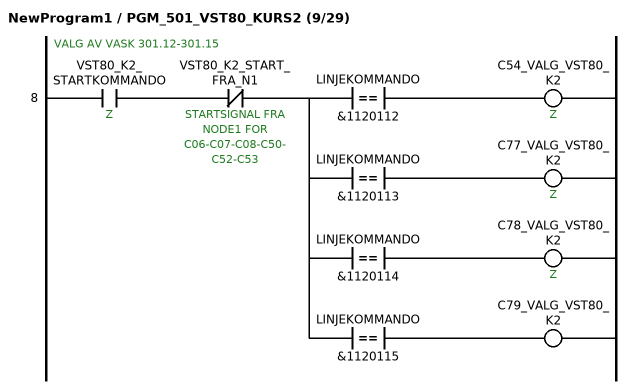
; [picture p504: NewProgram1 / PGM_501_VST80_KURS2, rungs 8-8]
; rung 8: VALG AV VASK 301.12-301.15
LD VST80_K2_STARTKOMMANDO  ; Z
ANDNOT VST80_K2_START_FRA_N1  ; STARTSIGNAL FRA NODE1 FOR C06-C07-C08-C50-C52-C53
OUT TR0
AND=L(301) LINJEKOMMANDO &1120112
OUT C54_VALG_VST80_K2  ; Z
LD TR0
AND=L(301) LINJEKOMMANDO &1120113
OUT C77_VALG_VST80_K2  ; Z
LD TR0
AND=L(301) LINJEKOMMANDO &1120114
OUT C78_VALG_VST80_K2  ; Z
LD TR0
AND=L(301) LINJEKOMMANDO &1120115
OUT C79_VALG_VST80_K2

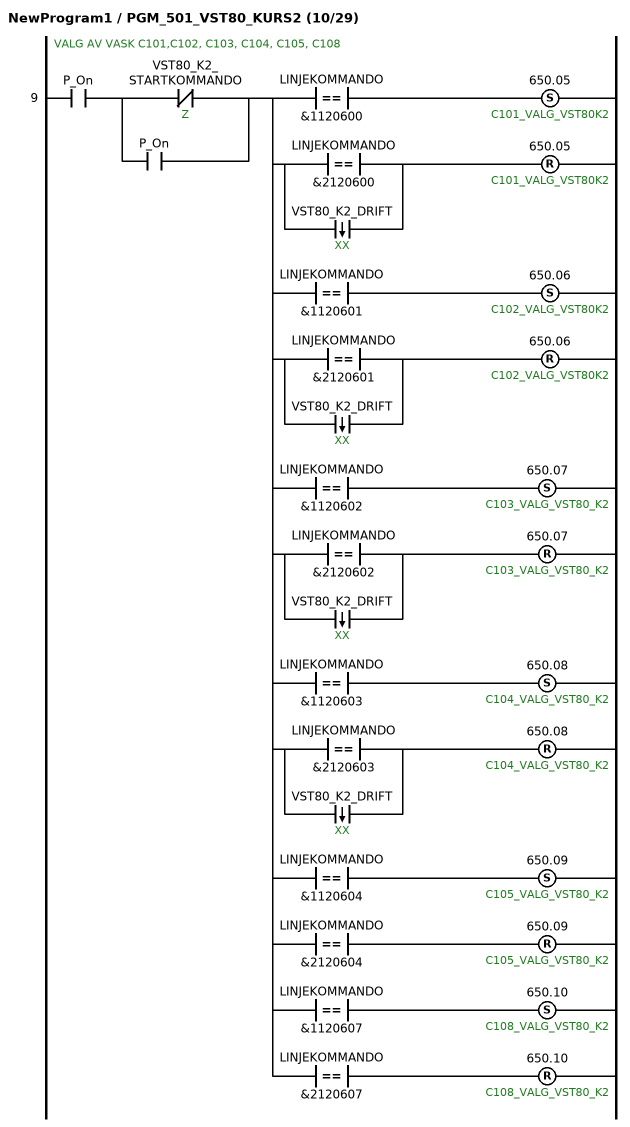
; rung 9: VALG AV VASK C101,C102, C103, C104, C105, C108
LD P_On
LDNOT VST80_K2_STARTKOMMANDO  ; Z
OR P_On
ANDLD
OUT TR0
AND=L(301) LINJEKOMMANDO &1120600
SET 650.05  ; C101_VALG_VST80K2
LD TR0
LD=L(301) LINJEKOMMANDO &2120600
%OR VST80_K2_DRIFT  ; XX
ANDLD
RSET 650.05  ; C101_VALG_VST80K2
LD TR0
AND=L(301) LINJEKOMMANDO &1120601
SET 650.06  ; C102_VALG_VST80K2
LD TR0
LD=L(301) LINJEKOMMANDO &2120601
%OR VST80_K2_DRIFT  ; XX
ANDLD
RSET 650.06  ; C102_VALG_VST80K2
LD TR0
AND=L(301) LINJEKOMMANDO &1120602
SET 650.07  ; C103_VALG_VST80_K2
LD TR0
LD=L(301) LINJEKOMMANDO &2120602
%OR VST80_K2_DRIFT  ; XX
ANDLD
RSET 650.07  ; C103_VALG_VST80_K2
LD TR0
AND=L(301) LINJEKOMMANDO &1120603
SET 650.08  ; C104_VALG_VST80_K2
LD TR0
LD=L(301) LINJEKOMMANDO &2120603
%OR VST80_K2_DRIFT  ; XX
ANDLD
RSET 650.08  ; C104_VALG_VST80_K2
LD TR0
AND=L(301) LINJEKOMMANDO &1120604
SET 650.09  ; C105_VALG_VST80_K2
LD TR0
AND=L(301) LINJEKOMMANDO &2120604
RSET 650.09  ; C105_VALG_VST80_K2
LD TR0
AND=L(301) LINJEKOMMANDO &1120607
SET 650.10  ; C108_VALG_VST80_K2
LD TR0
AND=L(301) LINJEKOMMANDO &2120607
RSET 650.10  ; C108_VALG_VST80_K2

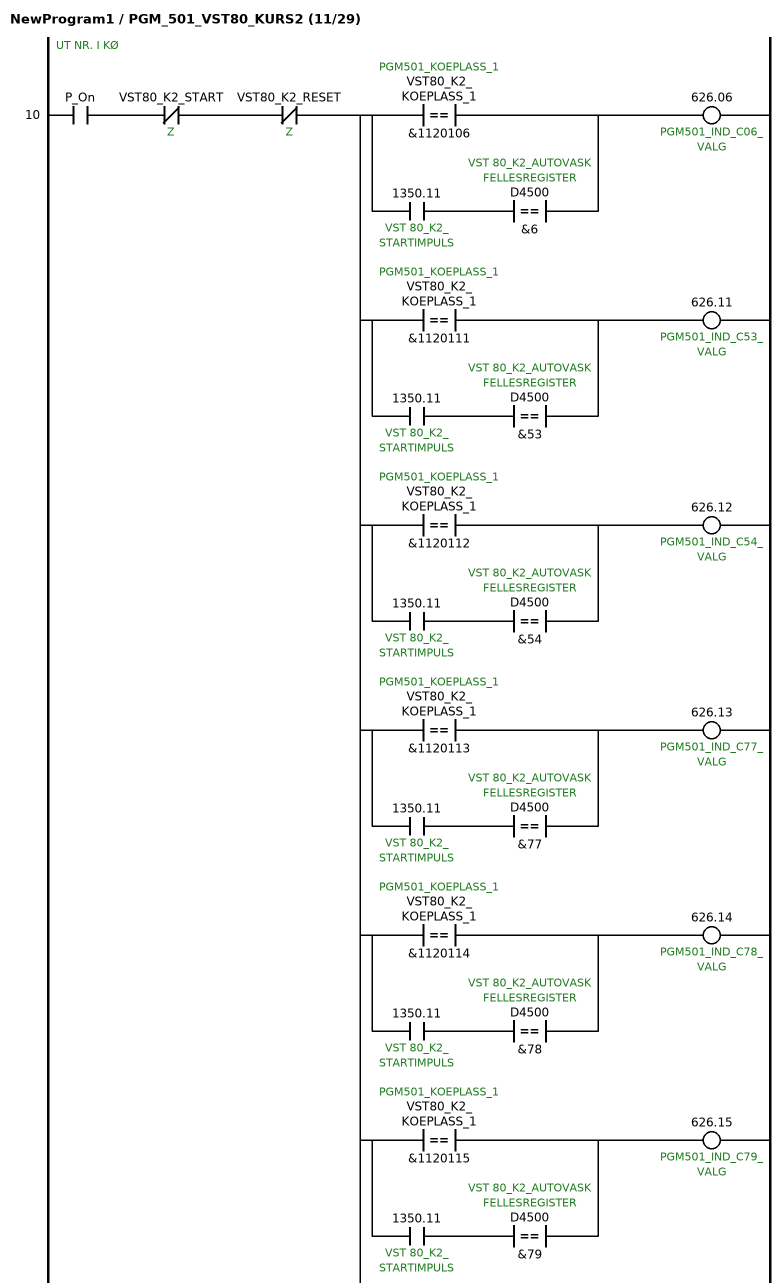

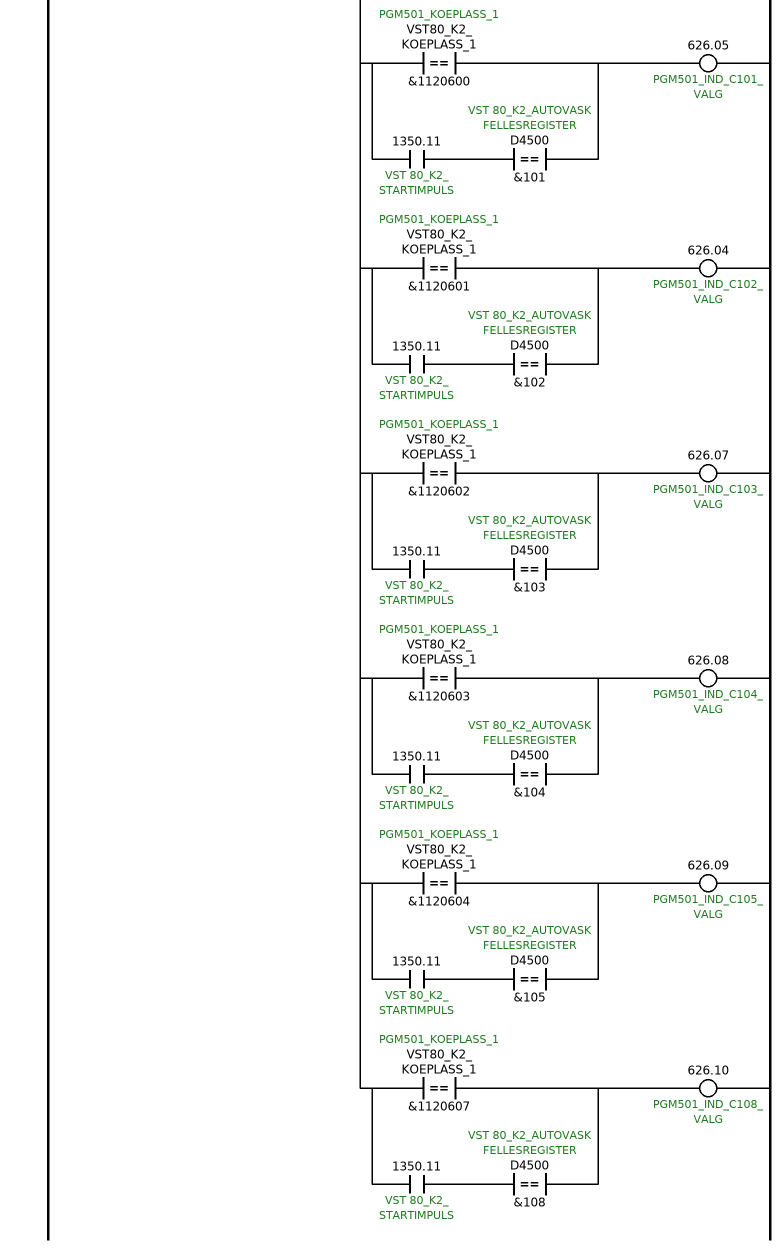
; rung 10: UT NR. I KØ
LD P_On
ANDNOT VST80_K2_START  ; Z
ANDNOT VST80_K2_RESET  ; Z
OUT TR0
LD=L(301) VST80_K2_KOEPLASS_1 &1120106  ; PGM501_KOEPLASS_1
LD 1350.11  ; VST 80_K2_STARTIMPULS
AND=(300) D4500 &6  ; VST 80_K2_AUTOVASK FELLESREGISTER
ORLD
ANDLD
OUT 626.06  ; PGM501_IND_C06_VALG
LD TR0
LD=L(301) VST80_K2_KOEPLASS_1 &1120111  ; PGM501_KOEPLASS_1
LD 1350.11  ; VST 80_K2_STARTIMPULS
AND=(300) D4500 &53  ; VST 80_K2_AUTOVASK FELLESREGISTER
ORLD
ANDLD
OUT 626.11  ; PGM501_IND_C53_VALG
LD TR0
LD=L(301) VST80_K2_KOEPLASS_1 &1120112  ; PGM501_KOEPLASS_1
LD 1350.11  ; VST 80_K2_STARTIMPULS
AND=(300) D4500 &54  ; VST 80_K2_AUTOVASK FELLESREGISTER
ORLD
ANDLD
OUT 626.12  ; PGM501_IND_C54_VALG
LD TR0
LD=L(301) VST80_K2_KOEPLASS_1 &1120113  ; PGM501_KOEPLASS_1
LD 1350.11  ; VST 80_K2_STARTIMPULS
AND=(300) D4500 &77  ; VST 80_K2_AUTOVASK FELLESREGISTER
ORLD
ANDLD
OUT 626.13  ; PGM501_IND_C77_VALG
LD TR0
LD=L(301) VST80_K2_KOEPLASS_1 &1120114  ; PGM501_KOEPLASS_1
LD 1350.11  ; VST 80_K2_STARTIMPULS
AND=(300) D4500 &78  ; VST 80_K2_AUTOVASK FELLESREGISTER
ORLD
ANDLD
OUT 626.14  ; PGM501_IND_C78_VALG
LD TR0
LD=L(301) VST80_K2_KOEPLASS_1 &1120115  ; PGM501_KOEPLASS_1
LD 1350.11  ; VST 80_K2_STARTIMPULS
AND=(300) D4500 &79  ; VST 80_K2_AUTOVASK FELLESREGISTER
ORLD
ANDLD
OUT 626.15  ; PGM501_IND_C79_VALG
LD TR0
LD=L(301) VST80_K2_KOEPLASS_1 &1120600  ; PGM501_KOEPLASS_1
LD 1350.11  ; VST 80_K2_STARTIMPULS
AND=(300) D4500 &101  ; VST 80_K2_AUTOVASK FELLESREGISTER
ORLD
ANDLD
OUT 626.05  ; PGM501_IND_C101_VALG
LD TR0
LD=L(301) VST80_K2_KOEPLASS_1 &1120601  ; PGM501_KOEPLASS_1
LD 1350.11  ; VST 80_K2_STARTIMPULS
AND=(300) D4500 &102  ; VST 80_K2_AUTOVASK FELLESREGISTER
ORLD
ANDLD
OUT 626.04  ; PGM501_IND_C102_VALG
LD TR0
LD=L(301) VST80_K2_KOEPLASS_1 &1120602  ; PGM501_KOEPLASS_1
LD 1350.11  ; VST 80_K2_STARTIMPULS
AND=(300) D4500 &103  ; VST 80_K2_AUTOVASK FELLESREGISTER
ORLD
ANDLD
OUT 626.07  ; PGM501_IND_C103_VALG
LD TR0
LD=L(301) VST80_K2_KOEPLASS_1 &1120603  ; PGM501_KOEPLASS_1
LD 1350.11  ; VST 80_K2_STARTIMPULS
AND=(300) D4500 &104  ; VST 80_K2_AUTOVASK FELLESREGISTER
ORLD
ANDLD
OUT 626.08  ; PGM501_IND_C104_VALG
LD TR0
LD=L(301) VST80_K2_KOEPLASS_1 &1120604  ; PGM501_KOEPLASS_1
LD 1350.11  ; VST 80_K2_STARTIMPULS
AND=(300) D4500 &105  ; VST 80_K2_AUTOVASK FELLESREGISTER
ORLD
ANDLD
OUT 626.09  ; PGM501_IND_C105_VALG
LD TR0
LD=L(301) VST80_K2_KOEPLASS_1 &1120607  ; PGM501_KOEPLASS_1
LD 1350.11  ; VST 80_K2_STARTIMPULS
AND=(300) D4500 &108  ; VST 80_K2_AUTOVASK FELLESREGISTER
ORLD
ANDLD
OUT 626.10  ; PGM501_IND_C108_VALG

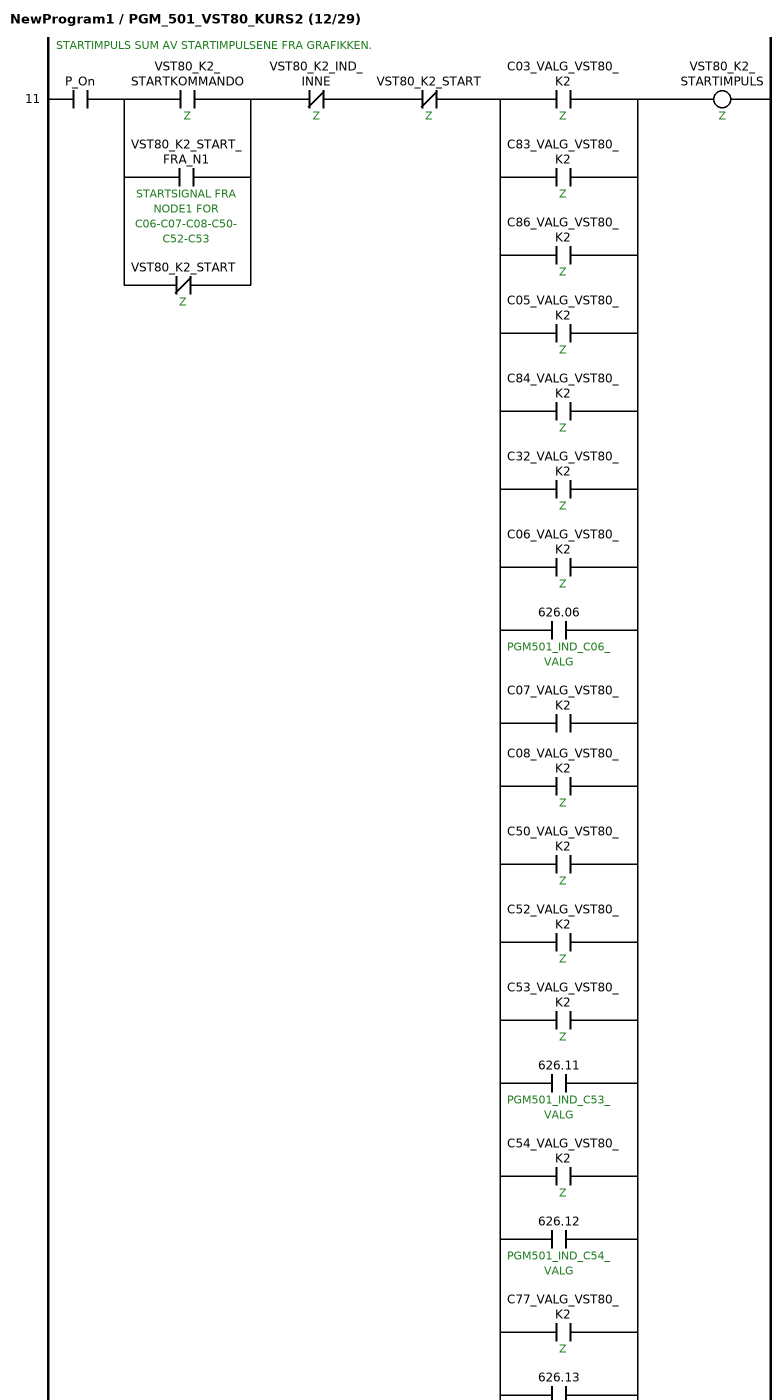

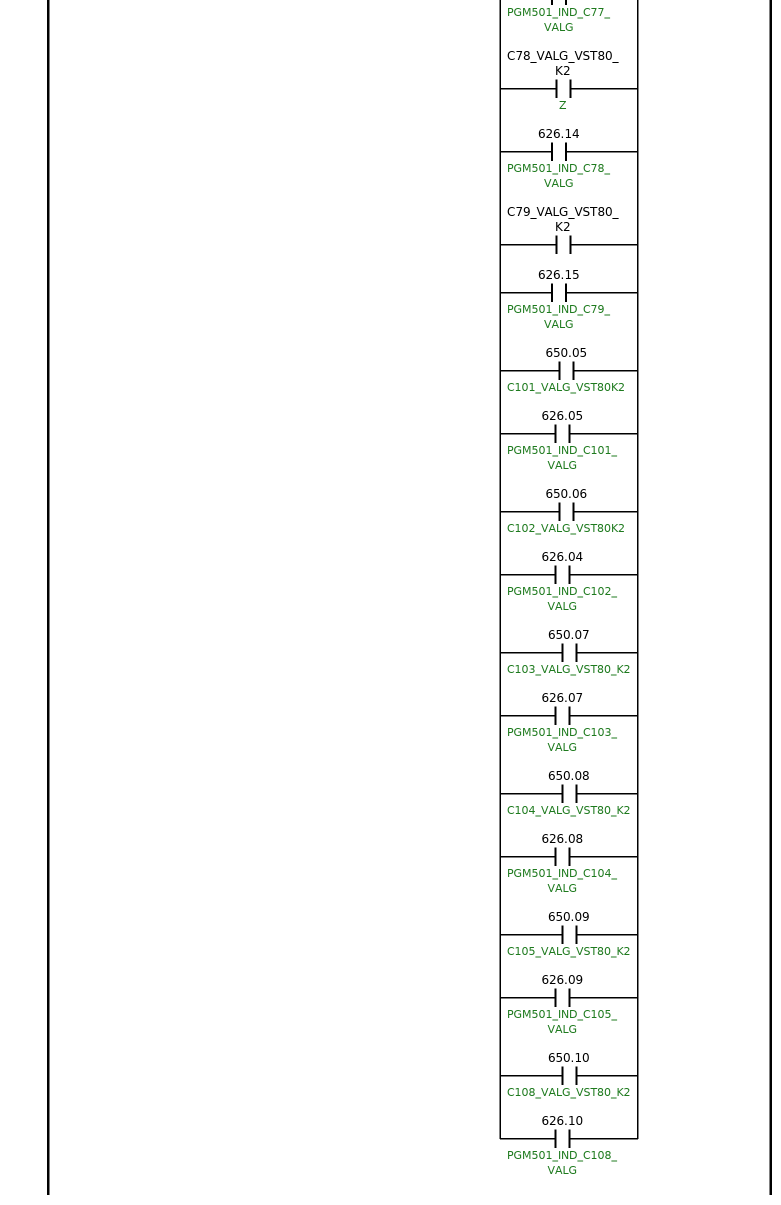
; rung 11: STARTIMPULS SUM AV STARTIMPULSENE FRA GRAFIKKEN.
LD P_On
LD VST80_K2_STARTKOMMANDO  ; Z
OR VST80_K2_START_FRA_N1  ; STARTSIGNAL FRA NODE1 FOR C06-C07-C08-C50-C52-C53
ORNOT VST80_K2_START  ; Z
ANDLD
ANDNOT VST80_K2_IND_INNE  ; Z
ANDNOT VST80_K2_START  ; Z
LD C03_VALG_VST80_K2  ; Z
OR C83_VALG_VST80_K2  ; Z
OR C86_VALG_VST80_K2  ; Z
OR C05_VALG_VST80_K2  ; Z
OR C84_VALG_VST80_K2  ; Z
OR C32_VALG_VST80_K2  ; Z
OR C06_VALG_VST80_K2  ; Z
OR 626.06  ; PGM501_IND_C06_VALG
OR C07_VALG_VST80_K2
OR C08_VALG_VST80_K2  ; Z
OR C50_VALG_VST80_K2  ; Z
OR C52_VALG_VST80_K2  ; Z
OR C53_VALG_VST80_K2  ; Z
OR 626.11  ; PGM501_IND_C53_VALG
OR C54_VALG_VST80_K2  ; Z
OR 626.12  ; PGM501_IND_C54_VALG
OR C77_VALG_VST80_K2  ; Z
OR 626.13  ; PGM501_IND_C77_VALG
OR C78_VALG_VST80_K2  ; Z
OR 626.14  ; PGM501_IND_C78_VALG
OR C79_VALG_VST80_K2
OR 626.15  ; PGM501_IND_C79_VALG
OR 650.05  ; C101_VALG_VST80K2
OR 626.05  ; PGM501_IND_C101_VALG
OR 650.06  ; C102_VALG_VST80K2
OR 626.04  ; PGM501_IND_C102_VALG
OR 650.07  ; C103_VALG_VST80_K2
OR 626.07  ; PGM501_IND_C103_VALG
OR 650.08  ; C104_VALG_VST80_K2
OR 626.08  ; PGM501_IND_C104_VALG
OR 650.09  ; C105_VALG_VST80_K2
OR 626.09  ; PGM501_IND_C105_VALG
OR 650.10  ; C108_VALG_VST80_K2
OR 626.10  ; PGM501_IND_C108_VALG
ANDLD
OUT VST80_K2_STARTIMPULS  ; Z

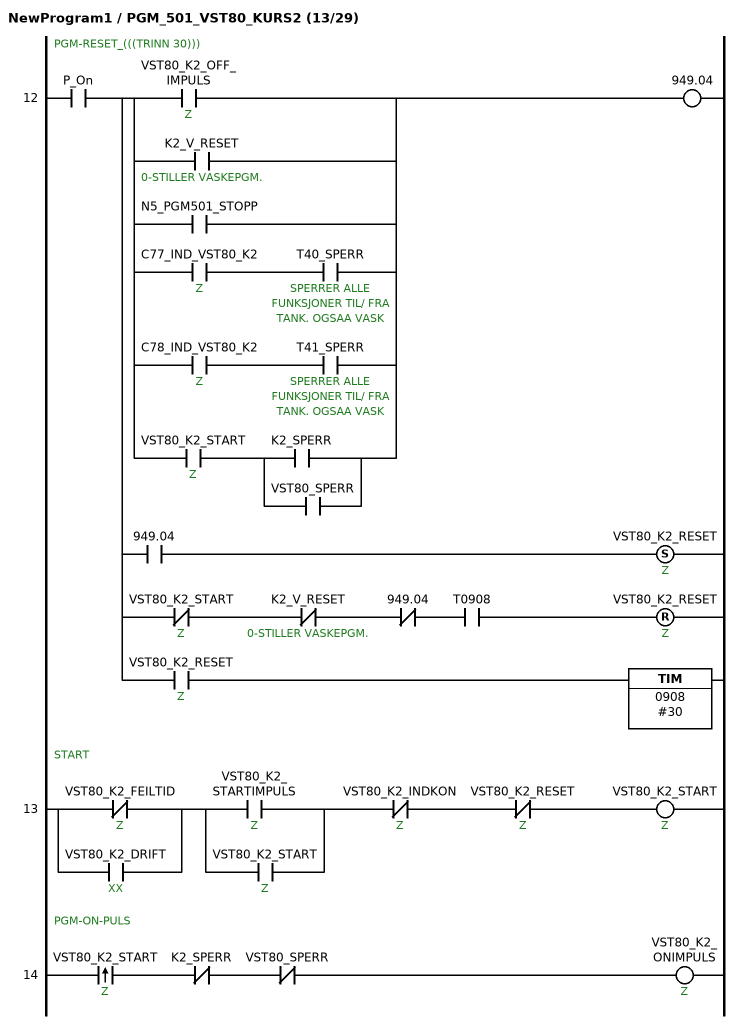
; rung 12: PGM-RESET_(((TRINN 30)))
LD P_On
OUT TR0
LD VST80_K2_OFF_IMPULS  ; Z
OR K2_V_RESET  ; 0-STILLER VASKEPGM.
OR N5_PGM501_STOPP
LD C77_IND_VST80_K2  ; Z
AND T40_SPERR  ; SPERRER ALLE FUNKSJONER TIL/ FRA TANK. OGSAA VASK
ORLD
LD C78_IND_VST80_K2  ; Z
AND T41_SPERR  ; SPERRER ALLE FUNKSJONER TIL/ FRA TANK. OGSAA VASK
ORLD
LD VST80_K2_START  ; Z
LD K2_SPERR
OR VST80_SPERR
ANDLD
ORLD
ANDLD
OUT 949.04
LD TR0
AND 949.04
SET VST80_K2_RESET  ; Z
LD TR0
ANDNOT VST80_K2_START  ; Z
ANDNOT K2_V_RESET  ; 0-STILLER VASKEPGM.
ANDNOT 949.04
AND T0908
RSET VST80_K2_RESET  ; Z
LD TR0
AND VST80_K2_RESET  ; Z
TIM 0908 #30
; rung 13: START
LDNOT VST80_K2_FEILTID  ; Z
OR VST80_K2_DRIFT  ; XX
LD VST80_K2_STARTIMPULS  ; Z
OR VST80_K2_START  ; Z
ANDLD
ANDNOT VST80_K2_INDKON  ; Z
ANDNOT VST80_K2_RESET  ; Z
OUT VST80_K2_START  ; Z
; rung 14: PGM-ON-PULS
@LD VST80_K2_START  ; Z
ANDNOT K2_SPERR
ANDNOT VST80_SPERR
OUT VST80_K2_ONIMPULS  ; Z

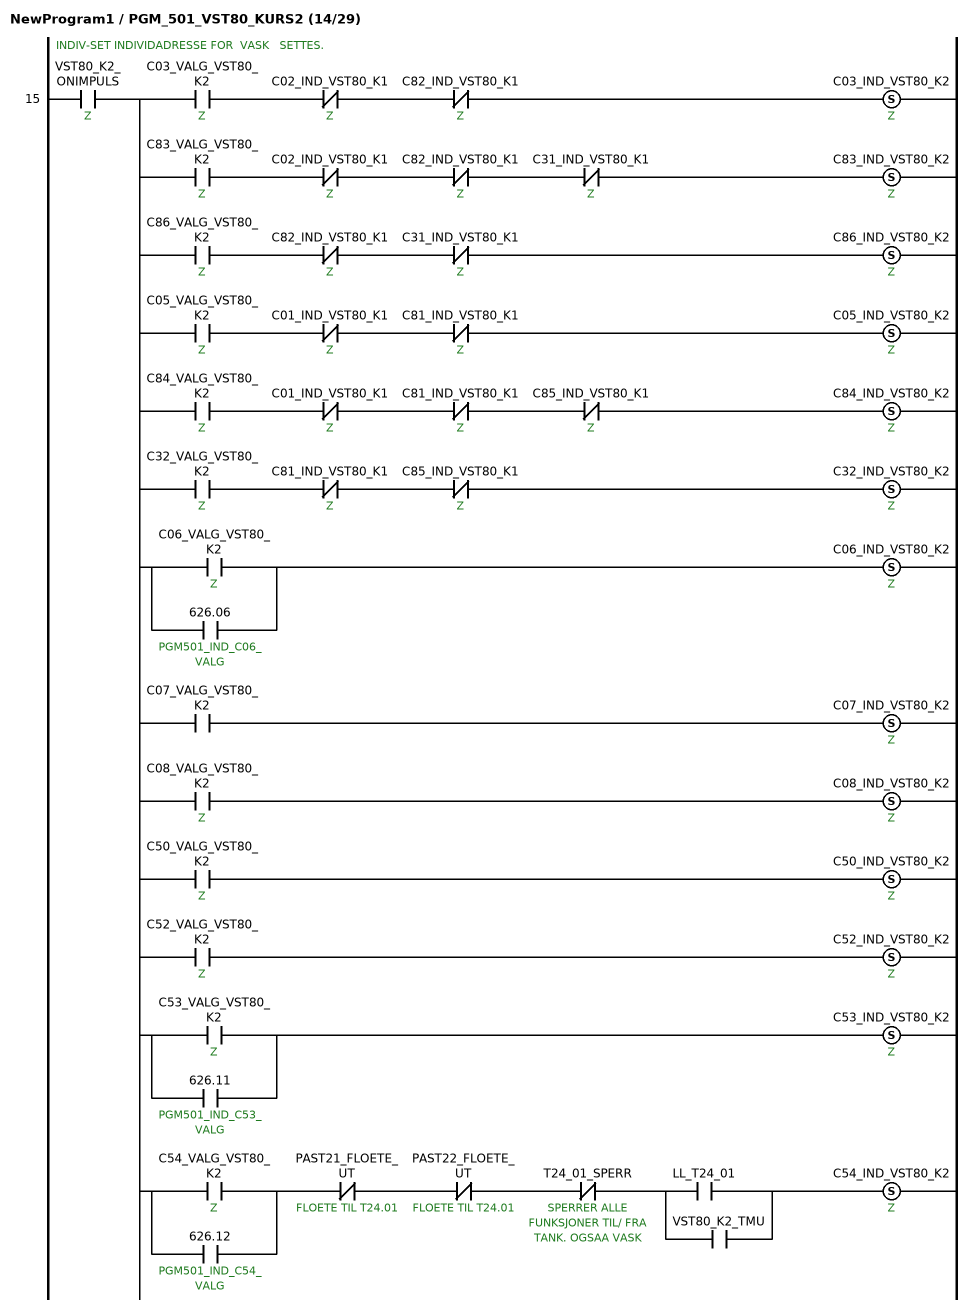

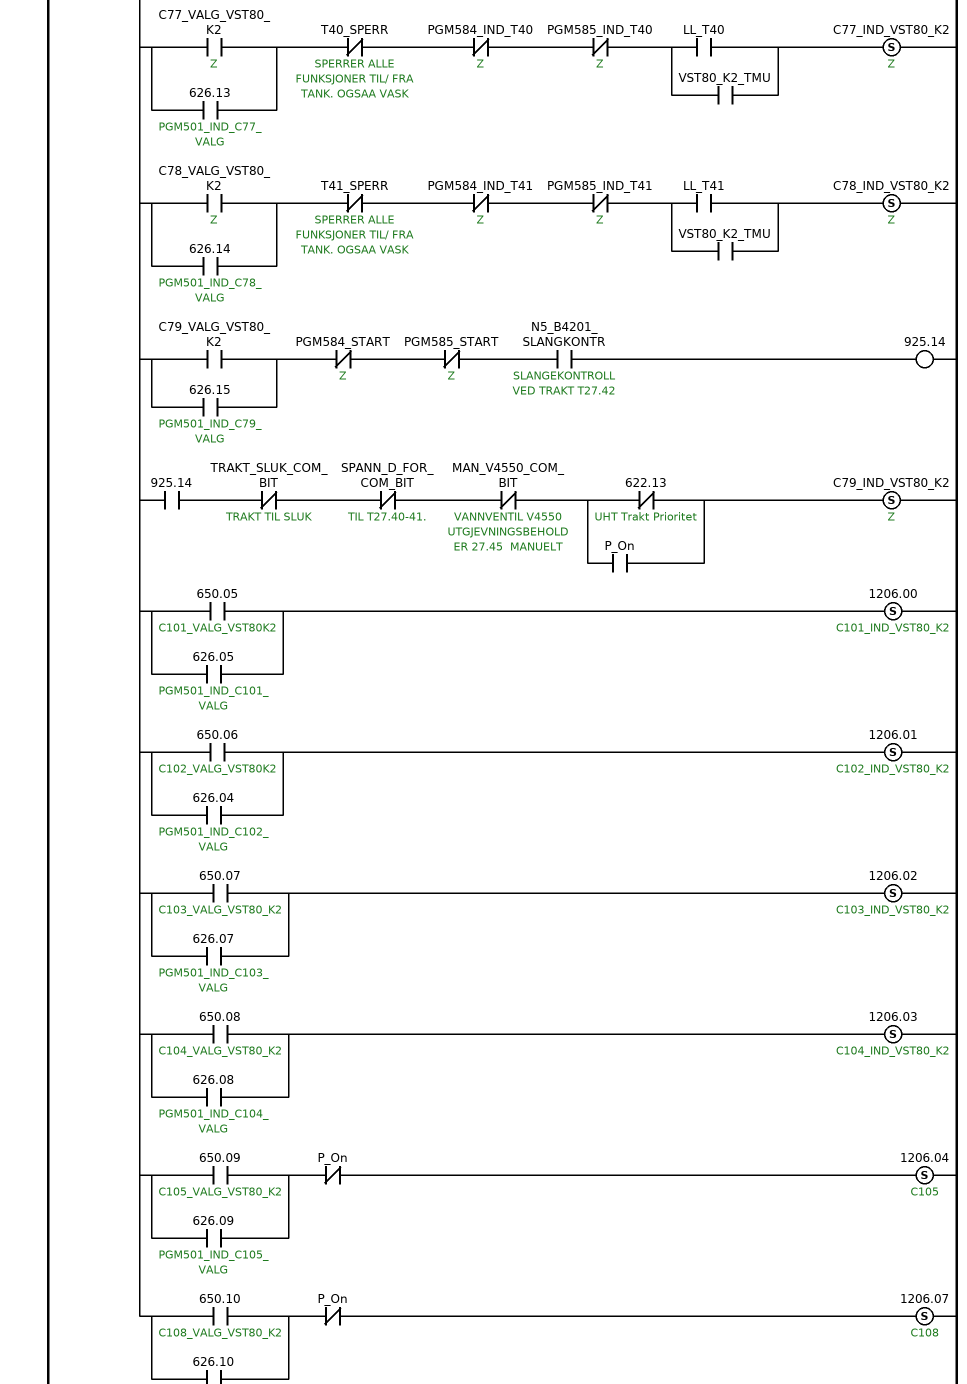

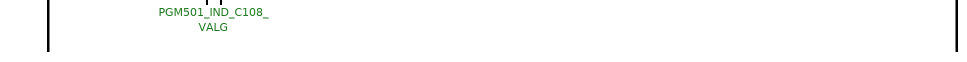
; rung 15: INDIV-SET INDIVIDADRESSE FOR  VASK   SETTES.
LD VST80_K2_ONIMPULS  ; Z
OUT TR0
AND C03_VALG_VST80_K2  ; Z
ANDNOT C02_IND_VST80_K1  ; Z
ANDNOT C82_IND_VST80_K1  ; Z
SET C03_IND_VST80_K2  ; Z
LD TR0
AND C83_VALG_VST80_K2  ; Z
ANDNOT C02_IND_VST80_K1  ; Z
ANDNOT C82_IND_VST80_K1  ; Z
ANDNOT C31_IND_VST80_K1  ; Z
SET C83_IND_VST80_K2  ; Z
LD TR0
AND C86_VALG_VST80_K2  ; Z
ANDNOT C82_IND_VST80_K1  ; Z
ANDNOT C31_IND_VST80_K1  ; Z
SET C86_IND_VST80_K2  ; Z
LD TR0
AND C05_VALG_VST80_K2  ; Z
ANDNOT C01_IND_VST80_K1  ; Z
ANDNOT C81_IND_VST80_K1  ; Z
SET C05_IND_VST80_K2  ; Z
LD TR0
AND C84_VALG_VST80_K2  ; Z
ANDNOT C01_IND_VST80_K1  ; Z
ANDNOT C81_IND_VST80_K1  ; Z
ANDNOT C85_IND_VST80_K1  ; Z
SET C84_IND_VST80_K2  ; Z
LD TR0
AND C32_VALG_VST80_K2  ; Z
ANDNOT C81_IND_VST80_K1  ; Z
ANDNOT C85_IND_VST80_K1  ; Z
SET C32_IND_VST80_K2  ; Z
LD TR0
LD C06_VALG_VST80_K2  ; Z
OR 626.06  ; PGM501_IND_C06_VALG
ANDLD
SET C06_IND_VST80_K2  ; Z
LD TR0
AND C07_VALG_VST80_K2
SET C07_IND_VST80_K2  ; Z
LD TR0
AND C08_VALG_VST80_K2  ; Z
SET C08_IND_VST80_K2  ; Z
LD TR0
AND C50_VALG_VST80_K2  ; Z
SET C50_IND_VST80_K2  ; Z
LD TR0
AND C52_VALG_VST80_K2  ; Z
SET C52_IND_VST80_K2  ; Z
LD TR0
LD C53_VALG_VST80_K2  ; Z
OR 626.11  ; PGM501_IND_C53_VALG
ANDLD
SET C53_IND_VST80_K2  ; Z
LD TR0
LD C54_VALG_VST80_K2  ; Z
OR 626.12  ; PGM501_IND_C54_VALG
ANDLD
ANDNOT PAST21_FLOETE_UT  ; FLOETE TIL T24.01
ANDNOT PAST22_FLOETE_UT  ; FLOETE TIL T24.01
ANDNOT T24_01_SPERR  ; SPERRER ALLE FUNKSJONER TIL/ FRA TANK. OGSAA VASK
LD LL_T24_01
OR VST80_K2_TMU
ANDLD
SET C54_IND_VST80_K2  ; Z
LD TR0
LD C77_VALG_VST80_K2  ; Z
OR 626.13  ; PGM501_IND_C77_VALG
ANDLD
ANDNOT T40_SPERR  ; SPERRER ALLE FUNKSJONER TIL/ FRA TANK. OGSAA VASK
ANDNOT PGM584_IND_T40  ; Z
ANDNOT PGM585_IND_T40  ; Z
LD LL_T40
OR VST80_K2_TMU
ANDLD
SET C77_IND_VST80_K2  ; Z
LD TR0
LD C78_VALG_VST80_K2  ; Z
OR 626.14  ; PGM501_IND_C78_VALG
ANDLD
ANDNOT T41_SPERR  ; SPERRER ALLE FUNKSJONER TIL/ FRA TANK. OGSAA VASK
ANDNOT PGM584_IND_T41  ; Z
ANDNOT PGM585_IND_T41  ; Z
LD LL_T41
OR VST80_K2_TMU
ANDLD
SET C78_IND_VST80_K2  ; Z
LD TR0
LD C79_VALG_VST80_K2
OR 626.15  ; PGM501_IND_C79_VALG
ANDLD
ANDNOT PGM584_START  ; Z
ANDNOT PGM585_START  ; Z
AND N5_B4201_SLANGKONTR  ; SLANGEKONTROLL VED TRAKT T27.42
OUT 925.14
LD TR0
AND 925.14
ANDNOT TRAKT_SLUK_COM_BIT  ; TRAKT TIL SLUK
ANDNOT SPANN_D_FOR_COM_BIT  ; TIL T27.40-41.
ANDNOT MAN_V4550_COM_BIT  ; VANNVENTIL V4550 UTGJEVNINGSBEHOLDER 27.45  MANUELT
LDNOT 622.13  ; UHT Trakt Prioritet
OR P_On
ANDLD
SET C79_IND_VST80_K2  ; Z
LD TR0
LD 650.05  ; C101_VALG_VST80K2
OR 626.05  ; PGM501_IND_C101_VALG
ANDLD
SET 1206.00  ; C101_IND_VST80_K2
LD TR0
LD 650.06  ; C102_VALG_VST80K2
OR 626.04  ; PGM501_IND_C102_VALG
ANDLD
SET 1206.01  ; C102_IND_VST80_K2
LD TR0
LD 650.07  ; C103_VALG_VST80_K2
OR 626.07  ; PGM501_IND_C103_VALG
ANDLD
SET 1206.02  ; C103_IND_VST80_K2
LD TR0
LD 650.08  ; C104_VALG_VST80_K2
OR 626.08  ; PGM501_IND_C104_VALG
ANDLD
SET 1206.03  ; C104_IND_VST80_K2
LD TR0
LD 650.09  ; C105_VALG_VST80_K2
OR 626.09  ; PGM501_IND_C105_VALG
ANDLD
ANDNOT P_On
SET 1206.04  ; C105
LD TR0
LD 650.10  ; C108_VALG_VST80_K2
OR 626.10  ; PGM501_IND_C108_VALG
ANDLD
ANDNOT P_On
SET 1206.07  ; C108

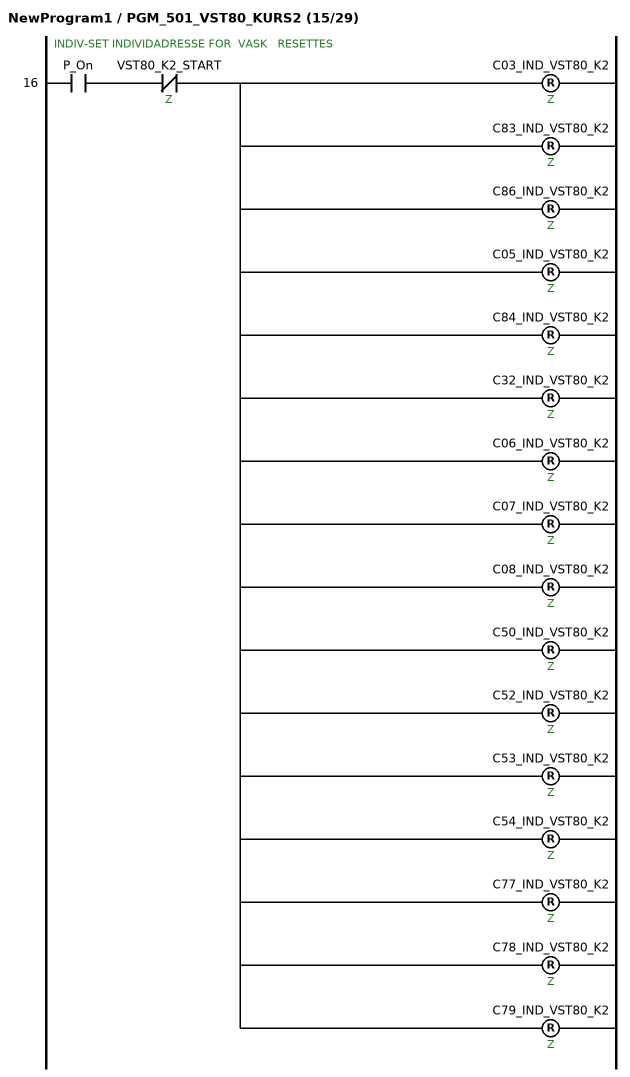
; rung 16: INDIV-SET INDIVIDADRESSE FOR  VASK   RESETTES
LD P_On
ANDNOT VST80_K2_START  ; Z
RSET C03_IND_VST80_K2  ; Z
RSET C83_IND_VST80_K2  ; Z
RSET C86_IND_VST80_K2  ; Z
RSET C05_IND_VST80_K2  ; Z
RSET C84_IND_VST80_K2  ; Z
RSET C32_IND_VST80_K2  ; Z
RSET C06_IND_VST80_K2  ; Z
RSET C07_IND_VST80_K2  ; Z
RSET C08_IND_VST80_K2  ; Z
RSET C50_IND_VST80_K2  ; Z
RSET C52_IND_VST80_K2  ; Z
RSET C53_IND_VST80_K2  ; Z
RSET C54_IND_VST80_K2  ; Z
RSET C77_IND_VST80_K2  ; Z
RSET C78_IND_VST80_K2  ; Z
RSET C79_IND_VST80_K2  ; Z

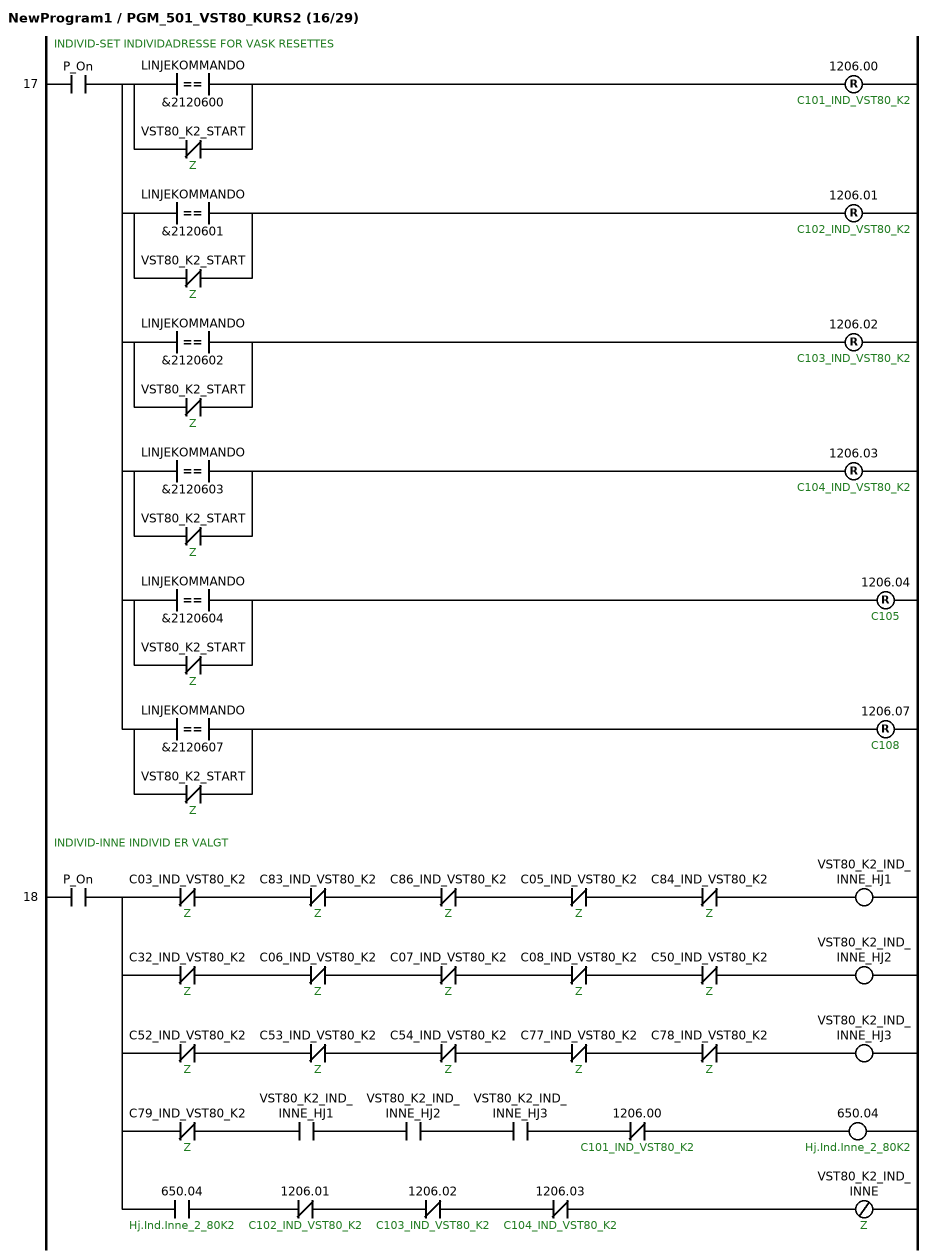
; rung 17: INDIVID-SET INDIVIDADRESSE FOR VASK RESETTES
LD P_On
OUT TR0
LD=L(301) LINJEKOMMANDO &2120600
ORNOT VST80_K2_START  ; Z
ANDLD
RSET 1206.00  ; C101_IND_VST80_K2
LD TR0
LD=L(301) LINJEKOMMANDO &2120601
ORNOT VST80_K2_START  ; Z
ANDLD
RSET 1206.01  ; C102_IND_VST80_K2
LD TR0
LD=L(301) LINJEKOMMANDO &2120602
ORNOT VST80_K2_START  ; Z
ANDLD
RSET 1206.02  ; C103_IND_VST80_K2
LD TR0
LD=L(301) LINJEKOMMANDO &2120603
ORNOT VST80_K2_START  ; Z
ANDLD
RSET 1206.03  ; C104_IND_VST80_K2
LD TR0
LD=L(301) LINJEKOMMANDO &2120604
ORNOT VST80_K2_START  ; Z
ANDLD
RSET 1206.04  ; C105
LD TR0
LD=L(301) LINJEKOMMANDO &2120607
ORNOT VST80_K2_START  ; Z
ANDLD
RSET 1206.07  ; C108
; rung 18: INDIVID-INNE INDIVID ER VALGT
LD P_On
OUT TR0
ANDNOT C03_IND_VST80_K2  ; Z
ANDNOT C83_IND_VST80_K2  ; Z
ANDNOT C86_IND_VST80_K2  ; Z
ANDNOT C05_IND_VST80_K2  ; Z
ANDNOT C84_IND_VST80_K2  ; Z
OUT VST80_K2_IND_INNE_HJ1
LD TR0
ANDNOT C32_IND_VST80_K2  ; Z
ANDNOT C06_IND_VST80_K2  ; Z
ANDNOT C07_IND_VST80_K2  ; Z
ANDNOT C08_IND_VST80_K2  ; Z
ANDNOT C50_IND_VST80_K2  ; Z
OUT VST80_K2_IND_INNE_HJ2
LD TR0
ANDNOT C52_IND_VST80_K2  ; Z
ANDNOT C53_IND_VST80_K2  ; Z
ANDNOT C54_IND_VST80_K2  ; Z
ANDNOT C77_IND_VST80_K2  ; Z
ANDNOT C78_IND_VST80_K2  ; Z
OUT VST80_K2_IND_INNE_HJ3
LD TR0
ANDNOT C79_IND_VST80_K2  ; Z
AND VST80_K2_IND_INNE_HJ1
AND VST80_K2_IND_INNE_HJ2
AND VST80_K2_IND_INNE_HJ3
ANDNOT 1206.00  ; C101_IND_VST80_K2
OUT 650.04  ; Hj.Ind.Inne_2_80K2
LD TR0
AND 650.04  ; Hj.Ind.Inne_2_80K2
ANDNOT 1206.01  ; C102_IND_VST80_K2
ANDNOT 1206.02  ; C103_IND_VST80_K2
ANDNOT 1206.03  ; C104_IND_VST80_K2
OUTNOT VST80_K2_IND_INNE  ; Z

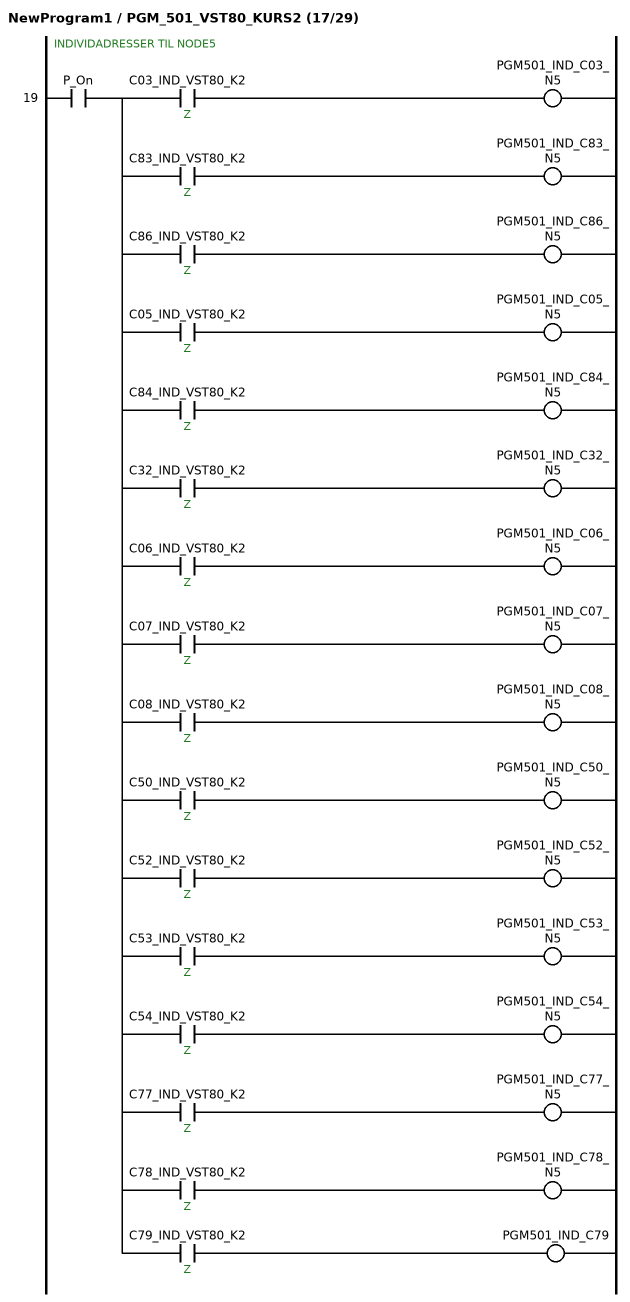
; rung 19: INDIVIDADRESSER TIL NODE5
LD P_On
OUT TR0
AND C03_IND_VST80_K2  ; Z
OUT PGM501_IND_C03_N5
LD TR0
AND C83_IND_VST80_K2  ; Z
OUT PGM501_IND_C83_N5
LD TR0
AND C86_IND_VST80_K2  ; Z
OUT PGM501_IND_C86_N5
LD TR0
AND C05_IND_VST80_K2  ; Z
OUT PGM501_IND_C05_N5
LD TR0
AND C84_IND_VST80_K2  ; Z
OUT PGM501_IND_C84_N5
LD TR0
AND C32_IND_VST80_K2  ; Z
OUT PGM501_IND_C32_N5
LD TR0
AND C06_IND_VST80_K2  ; Z
OUT PGM501_IND_C06_N5
LD TR0
AND C07_IND_VST80_K2  ; Z
OUT PGM501_IND_C07_N5
LD TR0
AND C08_IND_VST80_K2  ; Z
OUT PGM501_IND_C08_N5
LD TR0
AND C50_IND_VST80_K2  ; Z
OUT PGM501_IND_C50_N5
LD TR0
AND C52_IND_VST80_K2  ; Z
OUT PGM501_IND_C52_N5
LD TR0
AND C53_IND_VST80_K2  ; Z
OUT PGM501_IND_C53_N5
LD TR0
AND C54_IND_VST80_K2  ; Z
OUT PGM501_IND_C54_N5
LD TR0
AND C77_IND_VST80_K2  ; Z
OUT PGM501_IND_C77_N5
LD TR0
AND C78_IND_VST80_K2  ; Z
OUT PGM501_IND_C78_N5
LD TR0
AND C79_IND_VST80_K2  ; Z
OUT PGM501_IND_C79

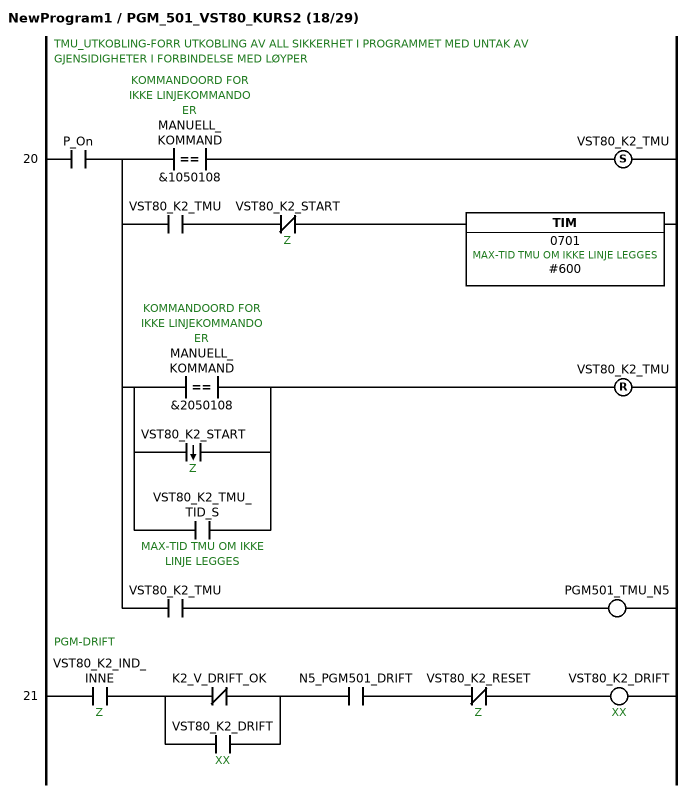
; rung 20: TMU_UTKOBLING-FORR UTKOBLING AV ALL SIKKERHET I PROGRAMMET MED UNTAK AV GJENSIDIGHETER I FORBINDELSE MED LØYPER
LD P_On
OUT TR0
AND=L(301) MANUELL_KOMMAND &1050108  ; KOMMANDOORD FOR IKKE LINJEKOMMANDOER
SET VST80_K2_TMU
LD TR0
AND VST80_K2_TMU
ANDNOT VST80_K2_START  ; Z
TIM 0701 #600  ; MAX-TID TMU OM IKKE LINJE LEGGES
LD TR0
LD=L(301) MANUELL_KOMMAND &2050108  ; KOMMANDOORD FOR IKKE LINJEKOMMANDOER
%OR VST80_K2_START  ; Z
OR VST80_K2_TMU_TID_S  ; MAX-TID TMU OM IKKE LINJE LEGGES
ANDLD
RSET VST80_K2_TMU
LD TR0
AND VST80_K2_TMU
OUT PGM501_TMU_N5
; rung 21: PGM-DRIFT
LD VST80_K2_IND_INNE  ; Z
LDNOT K2_V_DRIFT_OK
OR VST80_K2_DRIFT  ; XX
ANDLD
AND N5_PGM501_DRIFT
ANDNOT VST80_K2_RESET  ; Z
OUT VST80_K2_DRIFT  ; XX

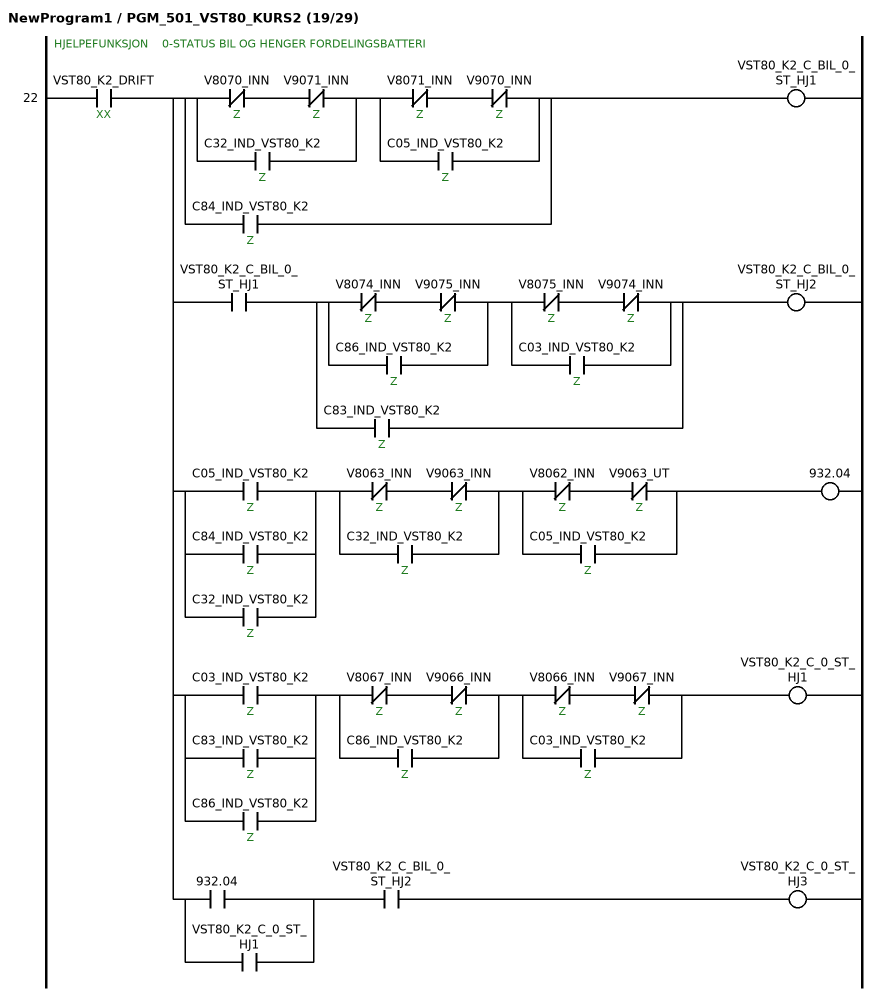
; rung 22: HJELPEFUNKSJON    0-STATUS BIL OG HENGER FORDELINGSBATTERI
LD VST80_K2_DRIFT  ; XX
OUT TR0
LDNOT V8070_INN  ; Z
ANDNOT V9071_INN  ; Z
OR C32_IND_VST80_K2  ; Z
LDNOT V8071_INN  ; Z
ANDNOT V9070_INN  ; Z
OR C05_IND_VST80_K2  ; Z
ANDLD
OR C84_IND_VST80_K2  ; Z
ANDLD
OUT VST80_K2_C_BIL_0_ST_HJ1
LD TR0
AND VST80_K2_C_BIL_0_ST_HJ1
LDNOT V8074_INN  ; Z
ANDNOT V9075_INN  ; Z
OR C86_IND_VST80_K2  ; Z
LDNOT V8075_INN  ; Z
ANDNOT V9074_INN  ; Z
OR C03_IND_VST80_K2  ; Z
ANDLD
OR C83_IND_VST80_K2  ; Z
ANDLD
OUT VST80_K2_C_BIL_0_ST_HJ2
LD TR0
LD C05_IND_VST80_K2  ; Z
OR C84_IND_VST80_K2  ; Z
OR C32_IND_VST80_K2  ; Z
ANDLD
LDNOT V8063_INN  ; Z
ANDNOT V9063_INN  ; Z
OR C32_IND_VST80_K2  ; Z
ANDLD
LDNOT V8062_INN  ; Z
ANDNOT V9063_UT  ; Z
OR C05_IND_VST80_K2  ; Z
ANDLD
OUT 932.04
LD TR0
LD C03_IND_VST80_K2  ; Z
OR C83_IND_VST80_K2  ; Z
OR C86_IND_VST80_K2  ; Z
ANDLD
LDNOT V8067_INN  ; Z
ANDNOT V9066_INN  ; Z
OR C86_IND_VST80_K2  ; Z
ANDLD
LDNOT V8066_INN  ; Z
ANDNOT V9067_INN  ; Z
OR C03_IND_VST80_K2  ; Z
ANDLD
OUT VST80_K2_C_0_ST_HJ1
LD TR0
LD 932.04
OR VST80_K2_C_0_ST_HJ1
ANDLD
AND VST80_K2_C_BIL_0_ST_HJ2
OUT VST80_K2_C_0_ST_HJ3

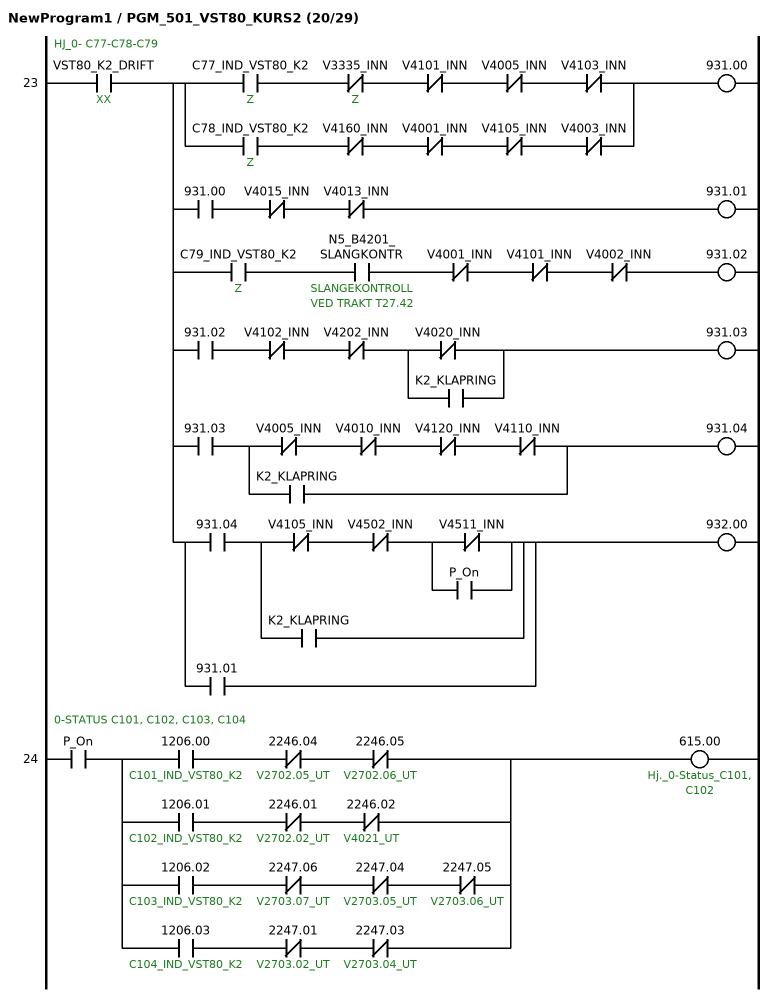
; rung 23: HJ_0- C77-C78-C79
LD VST80_K2_DRIFT  ; XX
OUT TR0
LD C77_IND_VST80_K2  ; Z
ANDNOT V3335_INN  ; Z
ANDNOT V4101_INN
ANDNOT V4005_INN
ANDNOT V4103_INN
LD C78_IND_VST80_K2  ; Z
ANDNOT V4160_INN
ANDNOT V4001_INN
ANDNOT V4105_INN
ANDNOT V4003_INN
ORLD
ANDLD
OUT 931.00
LD TR0
AND 931.00
ANDNOT V4015_INN
ANDNOT V4013_INN
OUT 931.01
LD TR0
AND C79_IND_VST80_K2  ; Z
AND N5_B4201_SLANGKONTR  ; SLANGEKONTROLL VED TRAKT T27.42
ANDNOT V4001_INN
ANDNOT V4101_INN
ANDNOT V4002_INN
OUT 931.02
LD TR0
AND 931.02
ANDNOT V4102_INN
ANDNOT V4202_INN
LDNOT V4020_INN
OR K2_KLAPRING
ANDLD
OUT 931.03
LD TR0
AND 931.03
LDNOT V4005_INN
ANDNOT V4010_INN
ANDNOT V4120_INN
ANDNOT V4110_INN
OR K2_KLAPRING
ANDLD
OUT 931.04
LD TR0
LD 931.04
LDNOT V4105_INN
ANDNOT V4502_INN
LDNOT V4511_INN
OR P_On
ANDLD
OR K2_KLAPRING
ANDLD
OR 931.01
ANDLD
OUT 932.00
; rung 24: 0-STATUS C101, C102, C103, C104
LD P_On
LD 1206.00  ; C101_IND_VST80_K2
ANDNOT 2246.04  ; V2702.05_UT
ANDNOT 2246.05  ; V2702.06_UT
LD 1206.01  ; C102_IND_VST80_K2
ANDNOT 2246.01  ; V2702.02_UT
ANDNOT 2246.02  ; V4021_UT
ORLD
LD 1206.02  ; C103_IND_VST80_K2
ANDNOT 2247.06  ; V2703.07_UT
ANDNOT 2247.04  ; V2703.05_UT
ANDNOT 2247.05  ; V2703.06_UT
ORLD
LD 1206.03  ; C104_IND_VST80_K2
ANDNOT 2247.01  ; V2703.02_UT
ANDNOT 2247.03  ; V2703.04_UT
ORLD
ANDLD
OUT 615.00  ; Hj._0-Status_C101,C102

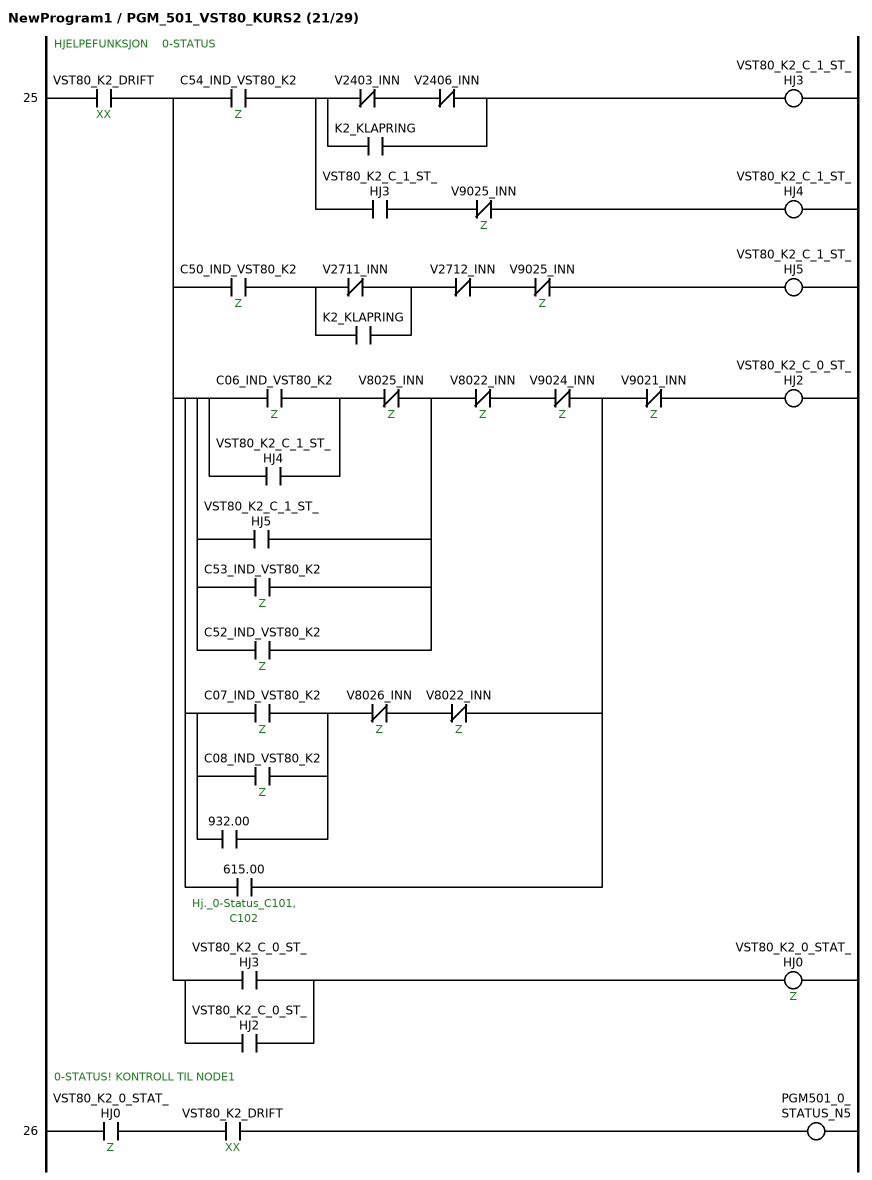
; rung 25: HJELPEFUNKSJON    0-STATUS
LD VST80_K2_DRIFT  ; XX
OUT TR0
AND C54_IND_VST80_K2  ; Z
OUT TR1
LDNOT V2403_INN
ANDNOT V2406_INN
OR K2_KLAPRING
ANDLD
OUT VST80_K2_C_1_ST_HJ3
LD TR1
AND VST80_K2_C_1_ST_HJ3
ANDNOT V9025_INN  ; Z
OUT VST80_K2_C_1_ST_HJ4
LD TR0
AND C50_IND_VST80_K2  ; Z
LDNOT V2711_INN
OR K2_KLAPRING
ANDLD
ANDNOT V2712_INN
ANDNOT V9025_INN  ; Z
OUT VST80_K2_C_1_ST_HJ5
LD TR0
LD C06_IND_VST80_K2  ; Z
OR VST80_K2_C_1_ST_HJ4
ANDNOT V8025_INN  ; Z
OR VST80_K2_C_1_ST_HJ5
OR C53_IND_VST80_K2  ; Z
OR C52_IND_VST80_K2  ; Z
ANDNOT V8022_INN  ; Z
ANDNOT V9024_INN  ; Z
LD C07_IND_VST80_K2  ; Z
OR C08_IND_VST80_K2  ; Z
OR 932.00
ANDNOT V8026_INN  ; Z
ANDNOT V8022_INN  ; Z
ORLD
OR 615.00  ; Hj._0-Status_C101,C102
ANDLD
ANDNOT V9021_INN  ; Z
OUT VST80_K2_C_0_ST_HJ2
LD TR0
LD VST80_K2_C_0_ST_HJ3
OR VST80_K2_C_0_ST_HJ2
ANDLD
OUT VST80_K2_0_STAT_HJ0  ; Z
; rung 26: 0-STATUS! KONTROLL TIL NODE1
LD VST80_K2_0_STAT_HJ0  ; Z
AND VST80_K2_DRIFT  ; XX
OUT PGM501_0_STATUS_N5

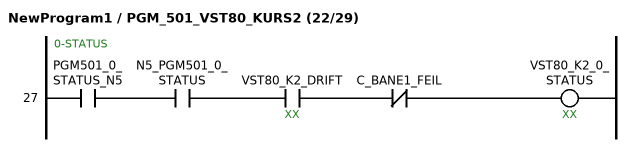
; rung 27: 0-STATUS
LD PGM501_0_STATUS_N5
AND N5_PGM501_0_STATUS
AND VST80_K2_DRIFT  ; XX
ANDNOT C_BANE1_FEIL
OUT VST80_K2_0_STATUS  ; XX

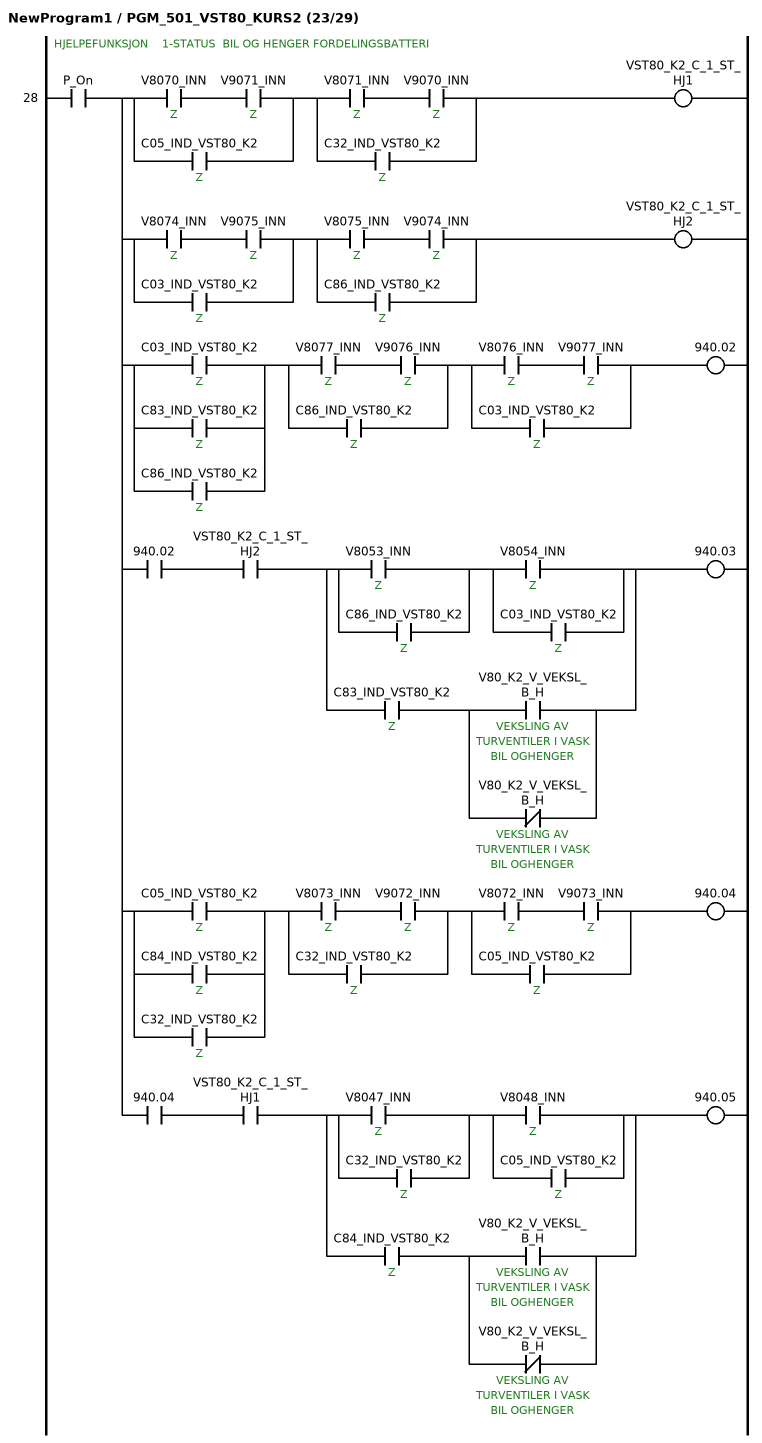
; rung 28: HJELPEFUNKSJON    1-STATUS  BIL OG HENGER FORDELINGSBATTERI
LD P_On
OUT TR0
LD V8070_INN  ; Z
AND V9071_INN  ; Z
OR C05_IND_VST80_K2  ; Z
ANDLD
LD V8071_INN  ; Z
AND V9070_INN  ; Z
OR C32_IND_VST80_K2  ; Z
ANDLD
OUT VST80_K2_C_1_ST_HJ1
LD TR0
LD V8074_INN  ; Z
AND V9075_INN  ; Z
OR C03_IND_VST80_K2  ; Z
ANDLD
LD V8075_INN  ; Z
AND V9074_INN  ; Z
OR C86_IND_VST80_K2  ; Z
ANDLD
OUT VST80_K2_C_1_ST_HJ2
LD TR0
LD C03_IND_VST80_K2  ; Z
OR C83_IND_VST80_K2  ; Z
OR C86_IND_VST80_K2  ; Z
ANDLD
LD V8077_INN  ; Z
AND V9076_INN  ; Z
OR C86_IND_VST80_K2  ; Z
ANDLD
LD V8076_INN  ; Z
AND V9077_INN  ; Z
OR C03_IND_VST80_K2  ; Z
ANDLD
OUT 940.02
LD TR0
AND 940.02
AND VST80_K2_C_1_ST_HJ2
LD V8053_INN  ; Z
OR C86_IND_VST80_K2  ; Z
LD V8054_INN  ; Z
OR C03_IND_VST80_K2  ; Z
ANDLD
LD C83_IND_VST80_K2  ; Z
LD V80_K2_V_VEKSL_B_H  ; VEKSLING AV TURVENTILER I VASK BIL OGHENGER
ORNOT V80_K2_V_VEKSL_B_H  ; VEKSLING AV TURVENTILER I VASK BIL OGHENGER
ANDLD
ORLD
ANDLD
OUT 940.03
LD TR0
LD C05_IND_VST80_K2  ; Z
OR C84_IND_VST80_K2  ; Z
OR C32_IND_VST80_K2  ; Z
ANDLD
LD V8073_INN  ; Z
AND V9072_INN  ; Z
OR C32_IND_VST80_K2  ; Z
ANDLD
LD V8072_INN  ; Z
AND V9073_INN  ; Z
OR C05_IND_VST80_K2  ; Z
ANDLD
OUT 940.04
LD TR0
AND 940.04
AND VST80_K2_C_1_ST_HJ1
LD V8047_INN  ; Z
OR C32_IND_VST80_K2  ; Z
LD V8048_INN  ; Z
OR C05_IND_VST80_K2  ; Z
ANDLD
LD C84_IND_VST80_K2  ; Z
LD V80_K2_V_VEKSL_B_H  ; VEKSLING AV TURVENTILER I VASK BIL OGHENGER
ORNOT V80_K2_V_VEKSL_B_H  ; VEKSLING AV TURVENTILER I VASK BIL OGHENGER
ANDLD
ORLD
ANDLD
OUT 940.05

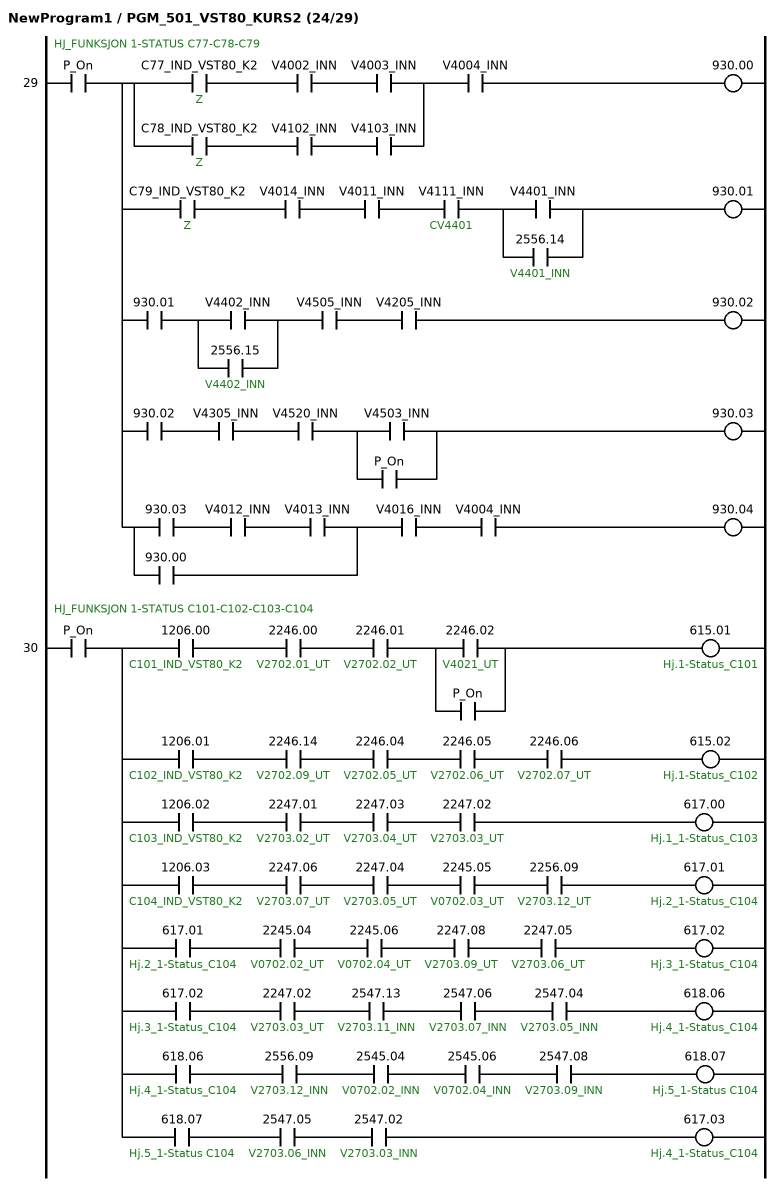
; rung 29: HJ_FUNKSJON 1-STATUS C77-C78-C79
LD P_On
OUT TR0
LD C77_IND_VST80_K2  ; Z
AND V4002_INN
AND V4003_INN
LD C78_IND_VST80_K2  ; Z
AND V4102_INN
AND V4103_INN
ORLD
ANDLD
AND V4004_INN
OUT 930.00
LD TR0
AND C79_IND_VST80_K2  ; Z
AND V4014_INN
AND V4011_INN
AND V4111_INN  ; CV4401
LD V4401_INN
OR 2556.14  ; V4401_INN
ANDLD
OUT 930.01
LD TR0
AND 930.01
LD V4402_INN
OR 2556.15  ; V4402_INN
ANDLD
AND V4505_INN
AND V4205_INN
OUT 930.02
LD TR0
AND 930.02
AND V4305_INN
AND V4520_INN
LD V4503_INN
OR P_On
ANDLD
OUT 930.03
LD TR0
LD 930.03
AND V4012_INN
AND V4013_INN
OR 930.00
ANDLD
AND V4016_INN
AND V4004_INN
OUT 930.04
; rung 30: HJ_FUNKSJON 1-STATUS C101-C102-C103-C104
LD P_On
OUT TR0
AND 1206.00  ; C101_IND_VST80_K2
AND 2246.00  ; V2702.01_UT
AND 2246.01  ; V2702.02_UT
LD 2246.02  ; V4021_UT
OR P_On
ANDLD
OUT 615.01  ; Hj.1-Status_C101
LD TR0
AND 1206.01  ; C102_IND_VST80_K2
AND 2246.14  ; V2702.09_UT
AND 2246.04  ; V2702.05_UT
AND 2246.05  ; V2702.06_UT
AND 2246.06  ; V2702.07_UT
OUT 615.02  ; Hj.1-Status_C102
LD TR0
AND 1206.02  ; C103_IND_VST80_K2
AND 2247.01  ; V2703.02_UT
AND 2247.03  ; V2703.04_UT
AND 2247.02  ; V2703.03_UT
OUT 617.00  ; Hj.1_1-Status_C103
LD TR0
AND 1206.03  ; C104_IND_VST80_K2
AND 2247.06  ; V2703.07_UT
AND 2247.04  ; V2703.05_UT
AND 2245.05  ; V0702.03_UT
AND 2256.09  ; V2703.12_UT
OUT 617.01  ; Hj.2_1-Status_C104
LD TR0
AND 617.01  ; Hj.2_1-Status_C104
AND 2245.04  ; V0702.02_UT
AND 2245.06  ; V0702.04_UT
AND 2247.08  ; V2703.09_UT
AND 2247.05  ; V2703.06_UT
OUT 617.02  ; Hj.3_1-Status_C104
LD TR0
AND 617.02  ; Hj.3_1-Status_C104
AND 2247.02  ; V2703.03_UT
AND 2547.13  ; V2703.11_INN
AND 2547.06  ; V2703.07_INN
AND 2547.04  ; V2703.05_INN
OUT 618.06  ; Hj.4_1-Status_C104
LD TR0
AND 618.06  ; Hj.4_1-Status_C104
AND 2556.09  ; V2703.12_INN
AND 2545.04  ; V0702.02_INN
AND 2545.06  ; V0702.04_INN
AND 2547.08  ; V2703.09_INN
OUT 618.07  ; Hj.5_1-Status C104
LD TR0
AND 618.07  ; Hj.5_1-Status C104
AND 2547.05  ; V2703.06_INN
AND 2547.02  ; V2703.03_INN
OUT 617.03  ; Hj.4_1-Status_C104

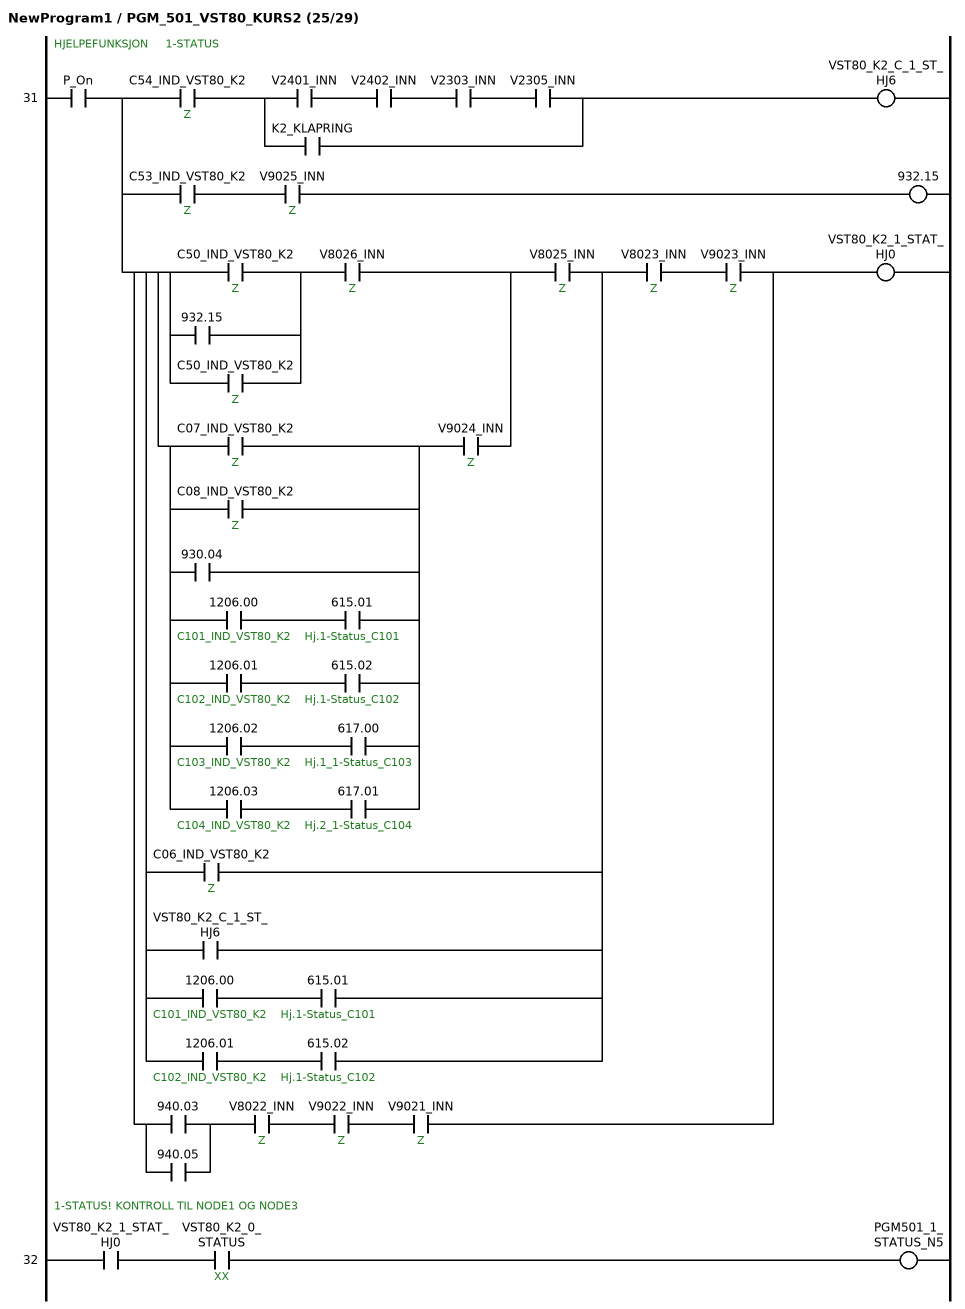
; rung 31: HJELPEFUNKSJON     1-STATUS
LD P_On
OUT TR0
AND C54_IND_VST80_K2  ; Z
LD V2401_INN
AND V2402_INN
AND V2303_INN
AND V2305_INN
OR K2_KLAPRING
ANDLD
OUT VST80_K2_C_1_ST_HJ6
LD TR0
AND C53_IND_VST80_K2  ; Z
AND V9025_INN  ; Z
OUT 932.15
LD TR0
LD C50_IND_VST80_K2  ; Z
OR 932.15
OR C50_IND_VST80_K2  ; Z
AND V8026_INN  ; Z
LD C07_IND_VST80_K2  ; Z
OR C08_IND_VST80_K2  ; Z
OR 930.04
LD 1206.00  ; C101_IND_VST80_K2
AND 615.01  ; Hj.1-Status_C101
ORLD
LD 1206.01  ; C102_IND_VST80_K2
AND 615.02  ; Hj.1-Status_C102
ORLD
LD 1206.02  ; C103_IND_VST80_K2
AND 617.00  ; Hj.1_1-Status_C103
ORLD
LD 1206.03  ; C104_IND_VST80_K2
AND 617.01  ; Hj.2_1-Status_C104
ORLD
AND V9024_INN  ; Z
ORLD
AND V8025_INN  ; Z
OR C06_IND_VST80_K2  ; Z
OR VST80_K2_C_1_ST_HJ6
LD 1206.00  ; C101_IND_VST80_K2
AND 615.01  ; Hj.1-Status_C101
ORLD
LD 1206.01  ; C102_IND_VST80_K2
AND 615.02  ; Hj.1-Status_C102
ORLD
AND V8023_INN  ; Z
AND V9023_INN  ; Z
LD 940.03
OR 940.05
AND V8022_INN  ; Z
AND V9022_INN  ; Z
AND V9021_INN  ; Z
ORLD
ANDLD
OUT VST80_K2_1_STAT_HJ0
; rung 32: 1-STATUS! KONTROLL TIL NODE1 OG NODE3
LD VST80_K2_1_STAT_HJ0
AND VST80_K2_0_STATUS  ; XX
OUT PGM501_1_STATUS_N5

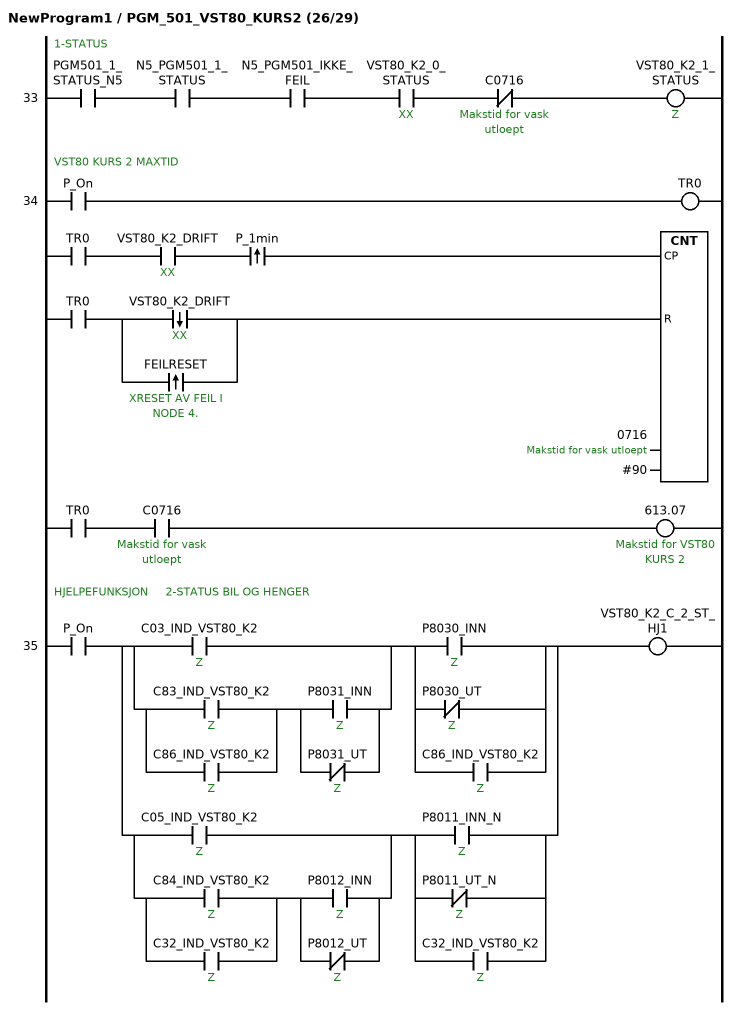
; rung 33: 1-STATUS
LD PGM501_1_STATUS_N5
AND N5_PGM501_1_STATUS
AND N5_PGM501_IKKE_FEIL
AND VST80_K2_0_STATUS  ; XX
ANDNOT C0716  ; Makstid for vask utloept
OUT VST80_K2_1_STATUS  ; Z
; rung 34: VST80 KURS 2 MAXTID
LD P_On
OUT TR0
AND VST80_K2_DRIFT  ; XX
@AND P_1min
LD TR0
%LD VST80_K2_DRIFT  ; XX
@OR FEILRESET  ; XRESET AV FEIL I NODE 4.
ANDLD
CNT 0716 #90  ; Makstid for vask utloept
LD TR0
AND C0716  ; Makstid for vask utloept
OUT 613.07  ; Makstid for VST80 KURS 2
; rung 35: HJELPEFUNKSJON     2-STATUS BIL OG HENGER
LD P_On
LD C03_IND_VST80_K2  ; Z
LD C83_IND_VST80_K2  ; Z
OR C86_IND_VST80_K2  ; Z
LD P8031_INN  ; Z
ORNOT P8031_UT  ; Z
ANDLD
ORLD
LD P8030_INN  ; Z
ORNOT P8030_UT  ; Z
OR C86_IND_VST80_K2  ; Z
ANDLD
LD C05_IND_VST80_K2  ; Z
LD C84_IND_VST80_K2  ; Z
OR C32_IND_VST80_K2  ; Z
LD P8012_INN  ; Z
ORNOT P8012_UT  ; Z
ANDLD
ORLD
LD P8011_INN_N  ; Z
ORNOT P8011_UT_N  ; Z
OR C32_IND_VST80_K2  ; Z
ANDLD
ORLD
ANDLD
OUT VST80_K2_C_2_ST_HJ1

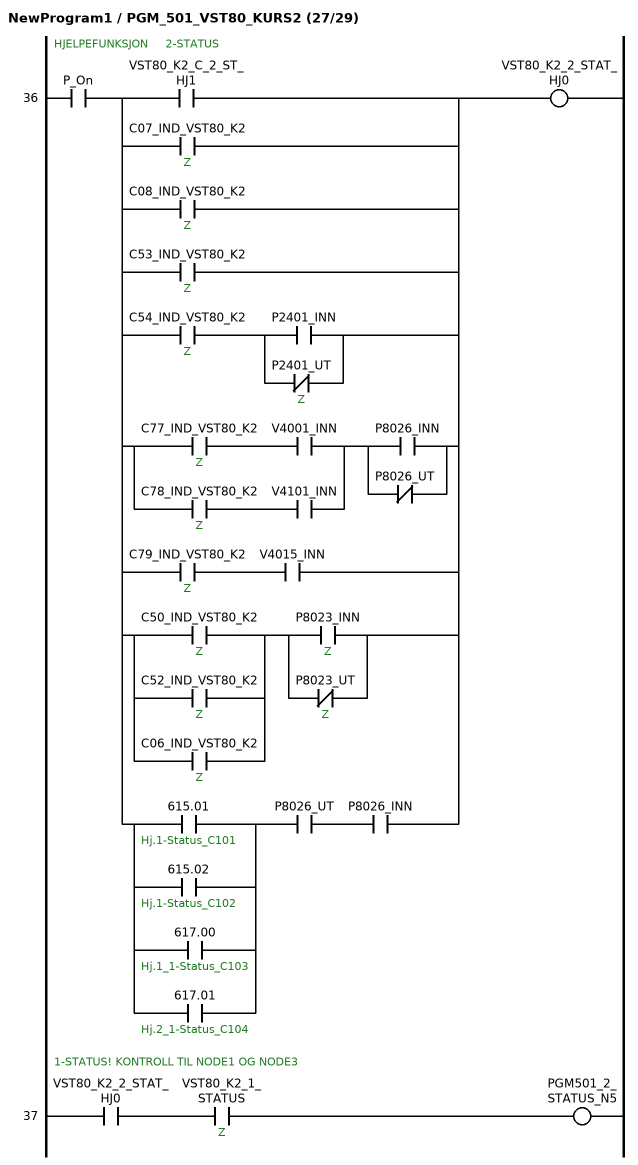
; rung 36: HJELPEFUNKSJON     2-STATUS
LD P_On
LD VST80_K2_C_2_ST_HJ1
OR C07_IND_VST80_K2  ; Z
OR C08_IND_VST80_K2  ; Z
OR C53_IND_VST80_K2  ; Z
LD C54_IND_VST80_K2  ; Z
LD P2401_INN
ORNOT P2401_UT  ; Z
ANDLD
ORLD
LD C77_IND_VST80_K2  ; Z
AND V4001_INN
LD C78_IND_VST80_K2  ; Z
AND V4101_INN
ORLD
LD P8026_INN
ORNOT P8026_UT
ANDLD
ORLD
LD C79_IND_VST80_K2  ; Z
AND V4015_INN
ORLD
LD C50_IND_VST80_K2  ; Z
OR C52_IND_VST80_K2  ; Z
OR C06_IND_VST80_K2  ; Z
LD P8023_INN  ; Z
ORNOT P8023_UT  ; Z
ANDLD
ORLD
LD 615.01  ; Hj.1-Status_C101
OR 615.02  ; Hj.1-Status_C102
OR 617.00  ; Hj.1_1-Status_C103
OR 617.01  ; Hj.2_1-Status_C104
AND P8026_UT
AND P8026_INN
ORLD
ANDLD
OUT VST80_K2_2_STAT_HJ0
; rung 37: 1-STATUS! KONTROLL TIL NODE1 OG NODE3
LD VST80_K2_2_STAT_HJ0
AND VST80_K2_1_STATUS  ; Z
OUT PGM501_2_STATUS_N5

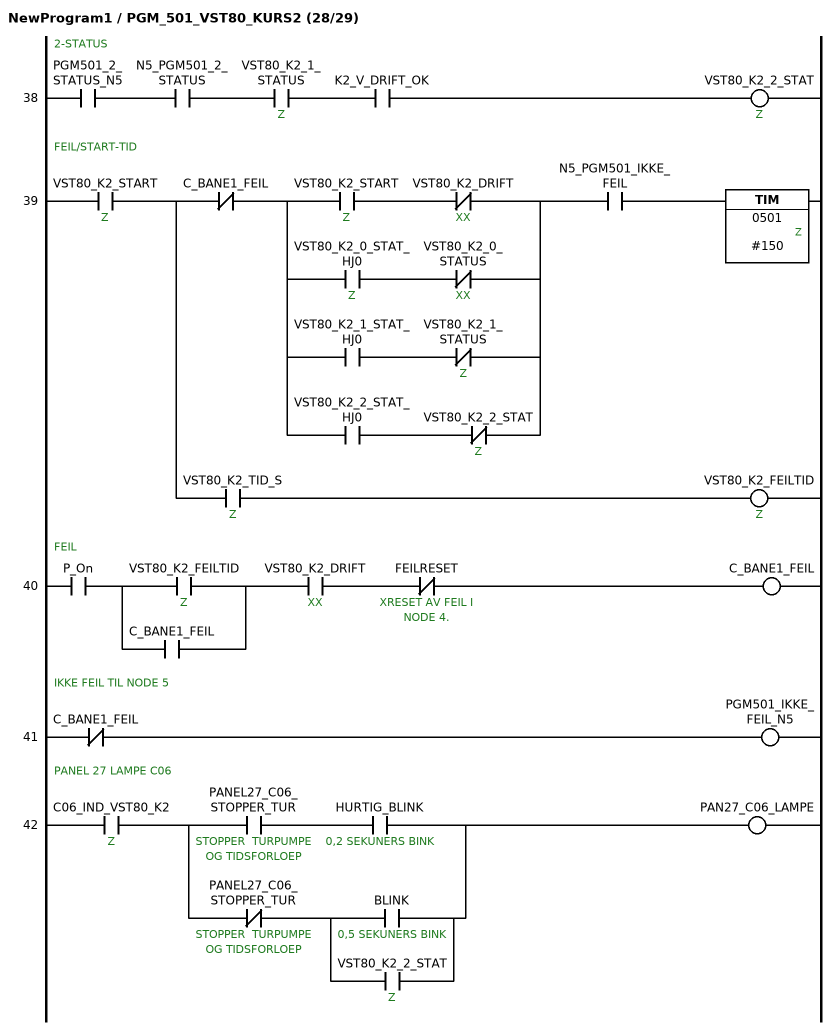
; rung 38: 2-STATUS
LD PGM501_2_STATUS_N5
AND N5_PGM501_2_STATUS
AND VST80_K2_1_STATUS  ; Z
AND K2_V_DRIFT_OK
OUT VST80_K2_2_STAT  ; Z
; rung 39: FEIL/START-TID
LD VST80_K2_START  ; Z
OUT TR0
ANDNOT C_BANE1_FEIL
LD VST80_K2_START  ; Z
ANDNOT VST80_K2_DRIFT  ; XX
LD VST80_K2_0_STAT_HJ0  ; Z
ANDNOT VST80_K2_0_STATUS  ; XX
ORLD
LD VST80_K2_1_STAT_HJ0
ANDNOT VST80_K2_1_STATUS  ; Z
ORLD
LD VST80_K2_2_STAT_HJ0
ANDNOT VST80_K2_2_STAT  ; Z
ORLD
ANDLD
AND N5_PGM501_IKKE_FEIL
TIM 0501 #150  ; Z
LD TR0
AND VST80_K2_TID_S  ; Z
OUT VST80_K2_FEILTID  ; Z
; rung 40: FEIL
LD P_On
LD VST80_K2_FEILTID  ; Z
OR C_BANE1_FEIL
ANDLD
AND VST80_K2_DRIFT  ; XX
ANDNOT FEILRESET  ; XRESET AV FEIL I NODE 4.
OUT C_BANE1_FEIL
; rung 41: IKKE FEIL TIL NODE 5
LDNOT C_BANE1_FEIL
OUT PGM501_IKKE_FEIL_N5
; rung 42: PANEL 27 LAMPE C06
LD C06_IND_VST80_K2  ; Z
LD PANEL27_C06_STOPPER_TUR  ; STOPPER  TURPUMPE OG TIDSFORLOEP
AND HURTIG_BLINK  ; 0,2 SEKUNERS BINK
LDNOT PANEL27_C06_STOPPER_TUR  ; STOPPER  TURPUMPE OG TIDSFORLOEP
LD BLINK  ; 0,5 SEKUNERS BINK
OR VST80_K2_2_STAT  ; Z
ANDLD
ORLD
ANDLD
OUT PAN27_C06_LAMPE

